VAR
	pAdress 		: PVOID;
	st_Variable		: ST_VarBuffer;
	bJson			: BOOL;
	tempString		: STRING;
	tempReal		: REAL;
	fbJson      	: FB_JsonSaxWriter;
	sJsonDocX12     : STRING(255);
	sJsonDocX11     : STRING(255);
	
	jsonKey			: STRING;
	i				: INT; // for loop index
	st_RW			: ST_RW;
END_VAR

VAR_OUTPUT
	sName			: STRING;
	eUpdate			: eUpdate;
	//bNumber		: BOOL;
	//bJson			: BOOL;
END_VAR
IF index < eDataMappingVarnames.last AND (aData[index].LogType = 0 OR aData[index].Label = '') THEN
	RETURN;
END_IF

CASE index OF 

//----(1)--- FILL STRUCTURES WITH DATA FROM PLC ------------------------------------------------------------
//----------------------------------------------------------------------------------------------------------
//--- eUpdate 0=Fast 1=Slow 2=Onchange 3=Daily--------------------------------------------------------------
//--- OnChange messages only get published when changing, at the same rate as the Fast timer----------------
//----st_Buffer contains properties of the given variable---------------------------------------------------
eDataMappingVarNames.safety_b_SafetyOK: 				st_Variable:= IotExtractType(monitor.safety.b_SafetyOK, 0, 0); 
eDataMappingVarNames.safety_b_EstopChannelAOK: 				st_Variable:= IotExtractType(monitor.safety.b_EstopChannelAOK, 0, 0); 
eDataMappingVarNames.safety_b_EstopChannelBOK: 				st_Variable:= IotExtractType(monitor.safety.b_EstopChannelBOK, 0, 0); 
eDataMappingVarNames.safety_b_InsulationMonitorOK: 				st_Variable:= IotExtractType(monitor.safety.b_InsulationMonitorOK, 0, 0); 
eDataMappingVarNames.safety_b_MRCDBOK: 				st_Variable:= IotExtractType(monitor.safety.b_MRCDBOK, 0, 0); 
// eDataMappingVarNames.safety_b_InverterDoorOK: 				st_Variable:= IotExtractType(monitor.safety.b_InverterDoorOK, 0, 0); 
// eDataMappingVarNames.safety_b_ZptOK: 				st_Variable:= IotExtractType(monitor.safety.b_ZptOK, 0, 0); 
// eDataMappingVarNames.system_b_SMSnumberConfigured: 				st_Variable:= IotExtractType(monitor.system.b_SMSnumberConfigured, 0, 0); 
// eDataMappingVarNames.system_b_CustomNameConfigured: 				st_Variable:= IotExtractType(monitor.system.b_CustomNameConfigured, 0, 0); 
// eDataMappingVarNames.system_s_SystemName: 				st_Variable:= IotExtractType(monitor.system.s_SystemName, 0, 0); 
// eDataMappingVarNames.system_b_TransportModePending: 				st_Variable:= IotExtractType(monitor.system.b_TransportModePending, 0, 0); 
// eDataMappingVarNames.system_b_DehumModePending: 				st_Variable:= IotExtractType(monitor.system.b_DehumModePending, 0, 0); 
// eDataMappingVarNames.system_e_State: 				st_Variable:= IotExtractType(monitor.system.e_State, 0, 0); 
// eDataMappingVarNames.system_e_gridmode: 				st_Variable:= IotExtractType(monitor.system.e_gridmode, 0, 0); 
// eDataMappingVarNames.system_e_UgridPowermode: 				st_Variable:= IotExtractType(monitor.system.e_UgridPowermode, 0, 0); 
// eDataMappingVarNames.system_b_StartAllowed: 				st_Variable:= IotExtractType(monitor.system.b_StartAllowed, 0, 0); 
// eDataMappingVarNames.system_r_CurrentEfficiency: 				st_Variable:= IotExtractType(monitor.system.r_CurrentEfficiency, 1, 0); 
// eDataMappingVarNames.system_r_AvgEfficiency: 				st_Variable:= IotExtractType(monitor.system.r_AvgEfficiency, 1, 0); 
// eDataMappingVarNames.system_r_RoundtripEfficiency: 				st_Variable:= IotExtractType(monitor.system.r_RoundtripEfficiency, 1, 0); 
// eDataMappingVarNames.system_DT_SystemTime: 				st_Variable:= IotExtractType(monitor.system.DT_SystemTime, 0, 0); 
// eDataMappingVarNames.system_PowerController_r_CurrentAct: 				st_Variable:= IotExtractType(monitor.system.PowerController.r_CurrentAct, 0, 1); 
// eDataMappingVarNames.system_PowerController_r_Sact: 				st_Variable:= IotExtractType(monitor.system.PowerController.r_Sact, 0, 1); 
// eDataMappingVarNames.system_PowerController_r_PAct: 				st_Variable:= IotExtractType(monitor.system.PowerController.r_PAct, 0, 1); 
// eDataMappingVarNames.system_PowerController_r_QAct: 				st_Variable:= IotExtractType(monitor.system.PowerController.r_QAct, 0, 1); 
// eDataMappingVarNames.system_PowerController_r_PhaseVoltageAct: 				st_Variable:= IotExtractType(monitor.system.PowerController.r_PhaseVoltageAct, 0, 1); 
// eDataMappingVarNames.system_PowerController_r_PFact: 				st_Variable:= IotExtractType(monitor.system.PowerController.r_PFact, 2, 0); 
// eDataMappingVarNames.system_PowerController_r_FeedInCurrentLimitActual: 				st_Variable:= IotExtractType(monitor.system.PowerController.r_FeedInCurrentLimitActual, 0, 0); 
// eDataMappingVarNames.system_PowerController_r_SupplyInCurrentLimitActual: 				st_Variable:= IotExtractType(monitor.system.PowerController.r_SupplyInCurrentLimitActual, 0, 0); 
// eDataMappingVarNames.system_PowerController_b_ThrottlingActive: 				st_Variable:= IotExtractType(monitor.system.PowerController.b_ThrottlingActive, 0, 0); 
// eDataMappingVarNames.system_PowerController_ui_ThrottlingType: 				st_Variable:= IotExtractType(monitor.system.PowerController.ui_ThrottlingType, 0, 0); 
// eDataMappingVarNames.system_PowerController_events_b_ReactivePIDError: 				st_Variable:= IotExtractType(monitor.system.PowerController.events.b_ReactivePIDError, 0, 0); 
// eDataMappingVarNames.system_PowerController_events_b_ActivePIDError: 				st_Variable:= IotExtractType(monitor.system.PowerController.events.b_ActivePIDError, 0, 0); 
// eDataMappingVarNames.system_PowerController_events_b_FreqShiftPIDError: 				st_Variable:= IotExtractType(monitor.system.PowerController.events.b_FreqShiftPIDError, 0, 0); 
// eDataMappingVarNames.system_GenGridController_b_active: 				st_Variable:= IotExtractType(monitor.system.GenGridController.b_active, 0, 0); 
// eDataMappingVarNames.system_GenGridController_b_faultActive: 				st_Variable:= IotExtractType(monitor.system.GenGridController.b_faultActive, 0, 0); 
// eDataMappingVarNames.system_GenGridController_b_gensetHot: 				st_Variable:= IotExtractType(monitor.system.GenGridController.b_gensetHot, 0, 0); 
// eDataMappingVarNames.system_GenGridController_b_gensetStarting: 				st_Variable:= IotExtractType(monitor.system.GenGridController.b_gensetStarting, 0, 0); 
// eDataMappingVarNames.system_GenGridController_b_ModeTransActive: 				st_Variable:= IotExtractType(monitor.system.GenGridController.b_ModeTransActive, 0, 0); 
// eDataMappingVarNames.system_GenGridController_b_ModeTransInhibit: 				st_Variable:= IotExtractType(monitor.system.GenGridController.b_ModeTransInhibit, 0, 0); 
// eDataMappingVarNames.system_GenGridController_b_ModeChanged: 				st_Variable:= IotExtractType(monitor.system.GenGridController.b_ModeChanged, 0, 0); 
// eDataMappingVarNames.system_GenGridController_b_ShowModeTrans: 				st_Variable:= IotExtractType(monitor.system.GenGridController.b_ShowModeTrans, 0, 0); 
// eDataMappingVarNames.system_GenGridController_b_extGensetMode: 				st_Variable:= IotExtractType(monitor.system.GenGridController.b_extGensetMode, 0, 0); 
// eDataMappingVarNames.system_GenGridController_b_gensetcontrol: 				st_Variable:= IotExtractType(monitor.system.GenGridController.b_gensetcontrol, 0, 0); 
// eDataMappingVarNames.system_GenGridController_e_BreakerMode: 				st_Variable:= IotExtractType(monitor.system.GenGridController.e_BreakerMode, 0, 0); 
// eDataMappingVarNames.system_GenGridController_e_PowerControlMode: 				st_Variable:= IotExtractType(monitor.system.GenGridController.e_PowerControlMode, 0, 0); 
// eDataMappingVarNames.system_GenGridController_e_GensetMode: 				st_Variable:= IotExtractType(monitor.system.GenGridController.e_GensetMode, 0, 0); 
// eDataMappingVarNames.system_GenGridController_e_GensetStartStop: 				st_Variable:= IotExtractType(monitor.system.GenGridController.e_GensetStartStop, 0, 0); 
// eDataMappingVarNames.system_GenGridController_e_state: 				st_Variable:= IotExtractType(monitor.system.GenGridController.e_state, 0, 0); 
// eDataMappingVarNames.system_GenGridController_e_RunCondition: 				st_Variable:= IotExtractType(monitor.system.GenGridController.e_RunCondition, 0, 0); 
// eDataMappingVarNames.system_GenGridController_events_b_InvalidGensetParameters: 				st_Variable:= IotExtractType(monitor.system.GenGridController.events.b_InvalidGensetParameters, 0, 0); 
// eDataMappingVarNames.system_GenGridController_events_b_RotationFieldFault: 				st_Variable:= IotExtractType(monitor.system.GenGridController.events.b_RotationFieldFault, 0, 0); 
// eDataMappingVarNames.system_GenGridController_events_b_CurrentLimitDisconnect: 				st_Variable:= IotExtractType(monitor.system.GenGridController.events.b_CurrentLimitDisconnect, 0, 0); 
// eDataMappingVarNames.system_GenGridController_events_b_CurrentLimitTrip: 				st_Variable:= IotExtractType(monitor.system.GenGridController.events.b_CurrentLimitTrip, 0, 0); 
// eDataMappingVarNames.system_GenGridController_events_b_EmstopDisconnect: 				st_Variable:= IotExtractType(monitor.system.GenGridController.events.b_EmstopDisconnect, 0, 0); 
// eDataMappingVarNames.system_GenGridController_events_b_ShutdownDisconnect: 				st_Variable:= IotExtractType(monitor.system.GenGridController.events.b_ShutdownDisconnect, 0, 0); 
// eDataMappingVarNames.system_GenGridController_events_b_OverloadTrip: 				st_Variable:= IotExtractType(monitor.system.GenGridController.events.b_OverloadTrip, 0, 0); 
// eDataMappingVarNames.system_GenGridController_events_b_OverFreqTrip: 				st_Variable:= IotExtractType(monitor.system.GenGridController.events.b_OverFreqTrip, 0, 0); 
// eDataMappingVarNames.system_GenGridController_events_b_UnderFreqTrip: 				st_Variable:= IotExtractType(monitor.system.GenGridController.events.b_UnderFreqTrip, 0, 0); 
// eDataMappingVarNames.system_GenGridController_events_b_OverVoltTrip: 				st_Variable:= IotExtractType(monitor.system.GenGridController.events.b_OverVoltTrip, 0, 0); 
// eDataMappingVarNames.system_GenGridController_events_b_UnderVoltTrip: 				st_Variable:= IotExtractType(monitor.system.GenGridController.events.b_UnderVoltTrip, 0, 0); 
// eDataMappingVarNames.system_GenGridController_events_b_ShutdownTimeOut: 				st_Variable:= IotExtractType(monitor.system.GenGridController.events.b_ShutdownTimeOut, 0, 0); 
// eDataMappingVarNames.system_GenGridController_events_b_SynchronisationFault: 				st_Variable:= IotExtractType(monitor.system.GenGridController.events.b_SynchronisationFault, 0, 0); 
// eDataMappingVarNames.system_GenGridController_events_b_StartupFault: 				st_Variable:= IotExtractType(monitor.system.GenGridController.events.b_StartupFault, 0, 0); 
// eDataMappingVarNames.system_GenGridController_events_b_WarmupFault: 				st_Variable:= IotExtractType(monitor.system.GenGridController.events.b_WarmupFault, 0, 0); 
// eDataMappingVarNames.system_GenGridController_events_b_GenDownTrip: 				st_Variable:= IotExtractType(monitor.system.GenGridController.events.b_GenDownTrip, 0, 0); 
// eDataMappingVarNames.system_GenGridController_events_b_GridLostTrip: 				st_Variable:= IotExtractType(monitor.system.GenGridController.events.b_GridLostTrip, 0, 0); 
// eDataMappingVarNames.system_GenGridController_events_b_TransToGenIsoInhibit: 				st_Variable:= IotExtractType(monitor.system.GenGridController.events.b_TransToGenIsoInhibit, 0, 0); 
// eDataMappingVarNames.system_GenGridController_events_b_TransToGenDroopInhibit: 				st_Variable:= IotExtractType(monitor.system.GenGridController.events.b_TransToGenDroopInhibit, 0, 0); 
// eDataMappingVarNames.system_GenGridController_events_b_TransToGenFixInhibit: 				st_Variable:= IotExtractType(monitor.system.GenGridController.events.b_TransToGenFixInhibit, 0, 0); 
// eDataMappingVarNames.system_GenGridController_events_b_TransFromInputGridAckRQ: 				st_Variable:= IotExtractType(monitor.system.GenGridController.events.b_TransFromInputGridAckRQ, 0, 0); 
// eDataMappingVarNames.system_GenGridController_events_b_TransFromInputGenAckRQ: 				st_Variable:= IotExtractType(monitor.system.GenGridController.events.b_TransFromInputGenAckRQ, 0, 0); 
// eDataMappingVarNames.system_GenGridController_events_b_StartingInhibit: 				st_Variable:= IotExtractType(monitor.system.GenGridController.events.b_StartingInhibit, 0, 0); 
// eDataMappingVarNames.system_events_b_RestartRequiredMachineName: 				st_Variable:= IotExtractType(monitor.system.events.b_RestartRequiredMachineName, 0, 0); 
// eDataMappingVarNames.system_events_b_TimeUpdateFailed: 				st_Variable:= IotExtractType(monitor.system.events.b_TimeUpdateFailed, 0, 0); 
// eDataMappingVarNames.powerstack_e_State: 				st_Variable:= IotExtractType(monitor.powerstack.e_State, 0, 0); 
// eDataMappingVarNames.powerstack_e_PowerState: 				st_Variable:= IotExtractType(monitor.powerstack.e_PowerState, 0, 0); 
// eDataMappingVarNames.powerstack_e_InverterMode: 				st_Variable:= IotExtractType(monitor.powerstack.e_InverterMode, 0, 0); 
// eDataMappingVarNames.powerstack_e_PowerMode: 				st_Variable:= IotExtractType(monitor.powerstack.e_PowerMode, 0, 0); 
// eDataMappingVarNames.powerstack_e_ThrottlingStatus: 				st_Variable:= IotExtractType(monitor.powerstack.e_ThrottlingStatus, 0, 0); 
// eDataMappingVarNames.powerstack_r_VoltageDroop: 				st_Variable:= IotExtractType(monitor.powerstack.r_VoltageDroop, 1, 0); 
// eDataMappingVarNames.powerstack_r_FrequencyDroop: 				st_Variable:= IotExtractType(monitor.powerstack.r_FrequencyDroop, 1, 0); 
// eDataMappingVarNames.powerstack_r_ACVoltageD7: 				st_Variable:= IotExtractType(monitor.powerstack.r_ACVoltageD7, 1, 1); 
// eDataMappingVarNames.powerstack_r_FrequencyD7: 				st_Variable:= IotExtractType(monitor.powerstack.r_FrequencyD7, 2, 1); 
// eDataMappingVarNames.powerstack_r_ActivePower: 				st_Variable:= IotExtractType(monitor.powerstack.r_ActivePower, 1, 1); 
// eDataMappingVarNames.powerstack_r_ReactivePower: 				st_Variable:= IotExtractType(monitor.powerstack.r_ReactivePower, 1, 1); 
// eDataMappingVarNames.powerstack_r_Pmin: 				st_Variable:= IotExtractType(monitor.powerstack.r_Pmin, 0, 0); 
// eDataMappingVarNames.powerstack_r_Pmax: 				st_Variable:= IotExtractType(monitor.powerstack.r_Pmax, 0, 0); 
// eDataMappingVarNames.powerstack_r_QMax: 				st_Variable:= IotExtractType(monitor.powerstack.r_QMax, 0, 0); 
// eDataMappingVarNames.powerstack_r_QMin: 				st_Variable:= IotExtractType(monitor.powerstack.r_QMin, 0, 0); 
// eDataMappingVarNames.powerstack_r_Smax: 				st_Variable:= IotExtractType(monitor.powerstack.r_Smax, 0, 0); 
// eDataMappingVarNames.powerstack_r_ACcurrentLimit: 				st_Variable:= IotExtractType(monitor.powerstack.r_ACcurrentLimit, 0, 0); 
// eDataMappingVarNames.powerstack_r_ACcurrentLimitMax: 				st_Variable:= IotExtractType(monitor.powerstack.r_ACcurrentLimitMax, 0, 0); 
// eDataMappingVarNames.powerstack_r_PowerChangeRate: 				st_Variable:= IotExtractType(monitor.powerstack.r_PowerChangeRate, 0, 0); 
// eDataMappingVarNames.powerstack_r_ApparentPower: 				st_Variable:= IotExtractType(monitor.powerstack.r_ApparentPower, 1, 1); 
// eDataMappingVarNames.powerstack_r_CosPhi: 				st_Variable:= IotExtractType(monitor.powerstack.r_CosPhi, 2, 0); 
// eDataMappingVarNames.powerstack_r_AcCurrent: 				st_Variable:= IotExtractType(monitor.powerstack.r_AcCurrent, 1, 0); 
// eDataMappingVarNames.powerstack_r_DCPower: 				st_Variable:= IotExtractType(monitor.powerstack.r_DCPower, 0, 1); 
// eDataMappingVarNames.powerstack_r_DCVoltage: 				st_Variable:= IotExtractType(monitor.powerstack.r_DCVoltage, 0, 1); 
// eDataMappingVarNames.powerstack_r_DCcurrent: 				st_Variable:= IotExtractType(monitor.powerstack.r_DCcurrent, 1, 1); 
// eDataMappingVarNames.powerstack_r_ACVoltageSupply: 				st_Variable:= IotExtractType(monitor.powerstack.r_ACVoltageSupply, 1, 1); 
// eDataMappingVarNames.powerstack_r_FrequencySupply: 				st_Variable:= IotExtractType(monitor.powerstack.r_FrequencySupply, 2, 1); 
// eDataMappingVarNames.powerstack_r_LoadPercent: 				st_Variable:= IotExtractType(monitor.powerstack.r_LoadPercent, 2, 0); 
// eDataMappingVarNames.powerstack_r_RatedCurrent: 				st_Variable:= IotExtractType(monitor.powerstack.r_RatedCurrent, 0, 0); 
// eDataMappingVarNames.powerstack_r_RatedPower: 				st_Variable:= IotExtractType(monitor.powerstack.r_RatedPower, 0, 0); 
// eDataMappingVarNames.powerstack_r_OvercurrentValueAct: 				st_Variable:= IotExtractType(monitor.powerstack.r_OvercurrentValueAct, 2, 0); 
// eDataMappingVarNames.powerstack_r_OvercurrentValueMax: 				st_Variable:= IotExtractType(monitor.powerstack.r_OvercurrentValueMax, 2, 0); 
// eDataMappingVarNames.powerstack_r_ThrottlingValueAct: 				st_Variable:= IotExtractType(monitor.powerstack.r_ThrottlingValueAct, 2, 0); 
// eDataMappingVarNames.powerstack_b_GridTied: 				st_Variable:= IotExtractType(monitor.powerstack.b_GridTied, 0, 0); 
// eDataMappingVarNames.powerstack_b_GridCodeCheckActive: 				st_Variable:= IotExtractType(monitor.powerstack.b_GridCodeCheckActive, 0, 0); 
// eDataMappingVarNames.powerstack_b_GridCodeOK: 				st_Variable:= IotExtractType(monitor.powerstack.b_GridCodeOK, 0, 0); 
// eDataMappingVarNames.powerstack_b_GridACdetected: 				st_Variable:= IotExtractType(monitor.powerstack.b_GridACdetected, 0, 0); 
// eDataMappingVarNames.powerstack_b_InverterGridFormingMode: 				st_Variable:= IotExtractType(monitor.powerstack.b_InverterGridFormingMode, 0, 0); 
// eDataMappingVarNames.powerstack_b_ACDetected: 				st_Variable:= IotExtractType(monitor.powerstack.b_ACDetected, 0, 0); 
// eDataMappingVarNames.powerstack_b_DCDetected: 				st_Variable:= IotExtractType(monitor.powerstack.b_DCDetected, 0, 0); 
// eDataMappingVarNames.powerstack_b_InverterRunning: 				st_Variable:= IotExtractType(monitor.powerstack.b_InverterRunning, 0, 0); 
// eDataMappingVarNames.powerstack_b_StartedState: 				st_Variable:= IotExtractType(monitor.powerstack.b_StartedState, 0, 0); 
// eDataMappingVarNames.powerstack_b_ControlEnabled: 				st_Variable:= IotExtractType(monitor.powerstack.b_ControlEnabled, 0, 0); 
// eDataMappingVarNames.powerstack_b_EcomodeAvailable: 				st_Variable:= IotExtractType(monitor.powerstack.b_EcomodeAvailable, 0, 0); 
// eDataMappingVarNames.powerstack_b_StartEnabled: 				st_Variable:= IotExtractType(monitor.powerstack.b_StartEnabled, 0, 0); 
// eDataMappingVarNames.powerstack_r_MaxTemperature: 				st_Variable:= IotExtractType(monitor.powerstack.r_MaxTemperature, 0, 0); 
// eDataMappingVarNames.powerstack_t_ShiftHoldTimeRemaining: 				st_Variable:= IotExtractType(monitor.powerstack.t_ShiftHoldTimeRemaining, 0, 0); 
// eDataMappingVarNames.powerstack_t_GridCodeReconnectTime: 				st_Variable:= IotExtractType(monitor.powerstack.t_GridCodeReconnectTime, 0, 0); 
// eDataMappingVarNames.powerstack_Events_b_CoolingDerating: 				st_Variable:= IotExtractType(monitor.powerstack.Events.b_CoolingDerating, 0, 0); 
// eDataMappingVarNames.powerstack_Events_b_PlimitShiftingActive: 				st_Variable:= IotExtractType(monitor.powerstack.Events.b_PlimitShiftingActive, 0, 0); 
// eDataMappingVarNames.powerstack_Events_b_DCdeviationHigh: 				st_Variable:= IotExtractType(monitor.powerstack.Events.b_DCdeviationHigh, 0, 0); 
// eDataMappingVarNames.powerstack_Events_b_TemperatureWarning: 				st_Variable:= IotExtractType(monitor.powerstack.Events.b_TemperatureWarning, 0, 0); 
// eDataMappingVarNames.powerstack_Events_b_OvercurrentWarning: 				st_Variable:= IotExtractType(monitor.powerstack.Events.b_OvercurrentWarning, 0, 0); 
// eDataMappingVarNames.powerstack_Events_b_UndervoltageWarning: 				st_Variable:= IotExtractType(monitor.powerstack.Events.b_UndervoltageWarning, 0, 0); 
// eDataMappingVarNames.powerstack_Events_b_OvervoltageWarning: 				st_Variable:= IotExtractType(monitor.powerstack.Events.b_OvervoltageWarning, 0, 0); 
// eDataMappingVarNames.powerstack_Events_b_TemperatureDeviationHigh: 				st_Variable:= IotExtractType(monitor.powerstack.Events.b_TemperatureDeviationHigh, 0, 0); 
// eDataMappingVarNames.powerstack_Events_b_PlimitShutdownWarning: 				st_Variable:= IotExtractType(monitor.powerstack.Events.b_PlimitShutdownWarning, 0, 0); 
// eDataMappingVarNames.powerstack_Events_b_MasterWarning: 				st_Variable:= IotExtractType(monitor.powerstack.Events.b_MasterWarning, 0, 0); 
// eDataMappingVarNames.powerstack_Events_b_SlaveWarning: 				st_Variable:= IotExtractType(monitor.powerstack.Events.b_SlaveWarning, 0, 0); 
// eDataMappingVarNames.powerstack_Events_b_GridCodeWarning: 				st_Variable:= IotExtractType(monitor.powerstack.Events.b_GridCodeWarning, 0, 0); 
// eDataMappingVarNames.powerstack_Events_b_UnderFreqFault: 				st_Variable:= IotExtractType(monitor.powerstack.Events.b_UnderFreqFault, 0, 0); 
// eDataMappingVarNames.powerstack_Events_b_OverFreqFault: 				st_Variable:= IotExtractType(monitor.powerstack.Events.b_OverFreqFault, 0, 0); 
// eDataMappingVarNames.powerstack_Events_b_UnderVoltageFault: 				st_Variable:= IotExtractType(monitor.powerstack.Events.b_UnderVoltageFault, 0, 0); 
// eDataMappingVarNames.powerstack_Events_b_OverVoltageFault: 				st_Variable:= IotExtractType(monitor.powerstack.Events.b_OverVoltageFault, 0, 0); 
// eDataMappingVarNames.powerstack_Events_b_OvercurrentFault: 				st_Variable:= IotExtractType(monitor.powerstack.Events.b_OvercurrentFault, 0, 0); 
// eDataMappingVarNames.powerstack_Events_b_PlimitShutdown: 				st_Variable:= IotExtractType(monitor.powerstack.Events.b_PlimitShutdown, 0, 0); 
// eDataMappingVarNames.powerstack_Events_b_TemperatureFault: 				st_Variable:= IotExtractType(monitor.powerstack.Events.b_TemperatureFault, 0, 0); 
// eDataMappingVarNames.powerstack_Events_b_MasterFault: 				st_Variable:= IotExtractType(monitor.powerstack.Events.b_MasterFault, 0, 0); 
// eDataMappingVarNames.powerstack_Events_b_SlaveFault: 				st_Variable:= IotExtractType(monitor.powerstack.Events.b_SlaveFault, 0, 0); 
// eDataMappingVarNames.powerstack_Events_b_NetcontactorFault: 				st_Variable:= IotExtractType(monitor.powerstack.Events.b_NetcontactorFault, 0, 0); 
// eDataMappingVarNames.powerstack_Events_b_startupTimeOut: 				st_Variable:= IotExtractType(monitor.powerstack.Events.b_startupTimeOut, 0, 0); 
// eDataMappingVarNames.powerstack_Events_b_ShutdownTimeOut: 				st_Variable:= IotExtractType(monitor.powerstack.Events.b_ShutdownTimeOut, 0, 0); 
// eDataMappingVarNames.powerstack_Events_ui_shutdownRemainingTime: 				st_Variable:= IotExtractType(monitor.powerstack.Events.ui_shutdownRemainingTime, 0, 0); 
// eDataMappingVarNames.powerstack_PowermoduleMaster_b_online: 				st_Variable:= IotExtractType(monitor.powerstack.PowermoduleMaster.b_online, 0, 0); 
// eDataMappingVarNames.powerstack_PowermoduleMaster_r_ApparentPower: 				st_Variable:= IotExtractType(monitor.powerstack.PowermoduleMaster.r_ApparentPower, 0, 1); 
// eDataMappingVarNames.powerstack_PowermoduleMaster_r_ActivePower: 				st_Variable:= IotExtractType(monitor.powerstack.PowermoduleMaster.r_ActivePower, 1, 1); 
// eDataMappingVarNames.powerstack_PowermoduleMaster_r_ReactivePower: 				st_Variable:= IotExtractType(monitor.powerstack.PowermoduleMaster.r_ReactivePower, 1, 1); 
// eDataMappingVarNames.powerstack_PowermoduleMaster_r_ACVoltageD7: 				st_Variable:= IotExtractType(monitor.powerstack.PowermoduleMaster.r_ACVoltageD7, 1, 1); 
// eDataMappingVarNames.powerstack_PowermoduleMaster_r_VoltageDroop: 				st_Variable:= IotExtractType(monitor.powerstack.PowermoduleMaster.r_VoltageDroop, 1, 0); 
// eDataMappingVarNames.powerstack_PowermoduleMaster_r_ACVoltageSupply: 				st_Variable:= IotExtractType(monitor.powerstack.PowermoduleMaster.r_ACVoltageSupply, 1, 1); 
// eDataMappingVarNames.powerstack_PowermoduleMaster_r_FrequencyD7: 				st_Variable:= IotExtractType(monitor.powerstack.PowermoduleMaster.r_FrequencyD7, 1, 1); 
// eDataMappingVarNames.powerstack_PowermoduleMaster_r_FrequencyDroop: 				st_Variable:= IotExtractType(monitor.powerstack.PowermoduleMaster.r_FrequencyDroop, 1, 0); 
// eDataMappingVarNames.powerstack_PowermoduleMaster_r_FrequencySupply: 				st_Variable:= IotExtractType(monitor.powerstack.PowermoduleMaster.r_FrequencySupply, 2, 1); 
// eDataMappingVarNames.powerstack_PowermoduleMaster_r_CurrentUnbalance: 				st_Variable:= IotExtractType(monitor.powerstack.PowermoduleMaster.r_CurrentUnbalance, 1, 1); 
// eDataMappingVarNames.powerstack_PowermoduleMaster_r_DCPower: 				st_Variable:= IotExtractType(monitor.powerstack.PowermoduleMaster.r_DCPower, 0, 1); 
// eDataMappingVarNames.powerstack_PowermoduleMaster_r_DCVoltage: 				st_Variable:= IotExtractType(monitor.powerstack.PowermoduleMaster.r_DCVoltage, 0, 1); 
// eDataMappingVarNames.powerstack_PowermoduleMaster_r_DCCurrent: 				st_Variable:= IotExtractType(monitor.powerstack.PowermoduleMaster.r_DCCurrent, 1, 0); 
// eDataMappingVarNames.powerstack_PowermoduleMaster_r_ACCurrent: 				st_Variable:= IotExtractType(monitor.powerstack.PowermoduleMaster.r_ACCurrent, 1, 1); 
// eDataMappingVarNames.powerstack_PowermoduleMaster_r_ActiveCurrent: 				st_Variable:= IotExtractType(monitor.powerstack.PowermoduleMaster.r_ActiveCurrent, 1, 1); 
// eDataMappingVarNames.powerstack_PowermoduleMaster_r_ReactiveCurrent: 				st_Variable:= IotExtractType(monitor.powerstack.PowermoduleMaster.r_ReactiveCurrent, 1, 1); 
// eDataMappingVarNames.powerstack_PowermoduleMaster_r_LoadPercent: 				st_Variable:= IotExtractType(monitor.powerstack.PowermoduleMaster.r_LoadPercent, 1, 0); 
// eDataMappingVarNames.powerstack_PowermoduleMaster_r_D7SyncError: 				st_Variable:= IotExtractType(monitor.powerstack.PowermoduleMaster.r_D7SyncError, 1, 0); 
// eDataMappingVarNames.powerstack_PowermoduleMaster_r_Pmin: 				st_Variable:= IotExtractType(monitor.powerstack.PowermoduleMaster.r_Pmin, 0, 0); 
// eDataMappingVarNames.powerstack_PowermoduleMaster_r_Pmax: 				st_Variable:= IotExtractType(monitor.powerstack.PowermoduleMaster.r_Pmax, 0, 0); 
// eDataMappingVarNames.powerstack_PowermoduleMaster_r_QMax: 				st_Variable:= IotExtractType(monitor.powerstack.PowermoduleMaster.r_QMax, 0, 0); 
// eDataMappingVarNames.powerstack_PowermoduleMaster_r_Qmin: 				st_Variable:= IotExtractType(monitor.powerstack.PowermoduleMaster.r_Qmin, 0, 0); 
// eDataMappingVarNames.powerstack_PowermoduleMaster_r_Pset: 				st_Variable:= IotExtractType(monitor.powerstack.PowermoduleMaster.r_Pset, 0, 0); 
// eDataMappingVarNames.powerstack_PowermoduleMaster_r_Qset: 				st_Variable:= IotExtractType(monitor.powerstack.PowermoduleMaster.r_Qset, 0, 0); 
// eDataMappingVarNames.powerstack_PowermoduleMaster_r_ACcurrentLimit: 				st_Variable:= IotExtractType(monitor.powerstack.PowermoduleMaster.r_ACcurrentLimit, 0, 0); 
// eDataMappingVarNames.powerstack_PowermoduleMaster_r_OverCurrentValue: 				st_Variable:= IotExtractType(monitor.powerstack.PowermoduleMaster.r_OverCurrentValue, 2, 0); 
// eDataMappingVarNames.powerstack_PowermoduleMaster_r_ModulationIndex: 				st_Variable:= IotExtractType(monitor.powerstack.PowermoduleMaster.r_ModulationIndex, 2, 0); 
// eDataMappingVarNames.powerstack_PowermoduleMaster_r_TemperatureInverter: 				st_Variable:= IotExtractType(monitor.powerstack.PowermoduleMaster.r_TemperatureInverter, 1, 0); 
// eDataMappingVarNames.powerstack_PowermoduleMaster_r_TemperatureGridChoke_1: 				st_Variable:= IotExtractType(monitor.powerstack.PowermoduleMaster.r_TemperatureGridChoke[1], 1, 0); 
// eDataMappingVarNames.powerstack_PowermoduleMaster_r_TemperatureGridChoke_2: 				st_Variable:= IotExtractType(monitor.powerstack.PowermoduleMaster.r_TemperatureGridChoke[2], 1, 0); 
// eDataMappingVarNames.powerstack_PowermoduleMaster_r_TemperatureGridChoke_3: 				st_Variable:= IotExtractType(monitor.powerstack.PowermoduleMaster.r_TemperatureGridChoke[3], 1, 0); 
// eDataMappingVarNames.powerstack_PowermoduleMaster_r_TemperatureCMChoke_1: 				st_Variable:= IotExtractType(monitor.powerstack.PowermoduleMaster.r_TemperatureCMChoke[1], 1, 0); 
// eDataMappingVarNames.powerstack_PowermoduleMaster_r_TemperatureCMChoke_2: 				st_Variable:= IotExtractType(monitor.powerstack.PowermoduleMaster.r_TemperatureCMChoke[2], 1, 0); 
// eDataMappingVarNames.powerstack_PowermoduleMaster_r_TemperatureCMChoke_3: 				st_Variable:= IotExtractType(monitor.powerstack.PowermoduleMaster.r_TemperatureCMChoke[3], 1, 0); 
// eDataMappingVarNames.powerstack_PowermoduleMaster_r_TemperatureCMChoke_4: 				st_Variable:= IotExtractType(monitor.powerstack.PowermoduleMaster.r_TemperatureCMChoke[4], 1, 0); 
// eDataMappingVarNames.powerstack_PowermoduleMaster_r_TemperatureMax: 				st_Variable:= IotExtractType(monitor.powerstack.PowermoduleMaster.r_TemperatureMax, 1, 0); 
// eDataMappingVarNames.powerstack_PowermoduleSlave_w_TemperatureFaultWord: 				st_Variable:= IotExtractType(monitor.powerstack.PowermoduleSlave.w_TemperatureFaultWord, 0, 0); 
// eDataMappingVarNames.powerstack_PowermoduleSlave_w_OperationHours: 				st_Variable:= IotExtractType(monitor.powerstack.PowermoduleSlave.w_OperationHours, 0, 0); 
// eDataMappingVarNames.powerstack_PowermoduleSlave_e_PowerMode: 				st_Variable:= IotExtractType(monitor.powerstack.PowermoduleSlave.e_PowerMode, 0, 0); 
// eDataMappingVarNames.powerstack_PowermoduleSlave_e_InverterMode: 				st_Variable:= IotExtractType(monitor.powerstack.PowermoduleSlave.e_InverterMode, 0, 0); 
// eDataMappingVarNames.powerstack_PowermoduleSlave_e_Status: 				st_Variable:= IotExtractType(monitor.powerstack.PowermoduleSlave.e_Status, 0, 0); 
// eDataMappingVarNames.powerstack_PowermoduleSlave_e_ThrottlingStatus: 				st_Variable:= IotExtractType(monitor.powerstack.PowermoduleSlave.e_ThrottlingStatus, 0, 0); 
// eDataMappingVarNames.powerstack_PowermoduleSlave_ui_InverterCommStatus: 				st_Variable:= IotExtractType(monitor.powerstack.PowermoduleSlave.ui_InverterCommStatus, 0, 0); 
// eDataMappingVarNames.powerstack_PowermoduleSlave_ui_BuscouplerCommStatus: 				st_Variable:= IotExtractType(monitor.powerstack.PowermoduleSlave.ui_BuscouplerCommStatus, 0, 0); 
// eDataMappingVarNames.powerstack_PowermoduleSlave_b_MccbTripOK: 				st_Variable:= IotExtractType(monitor.powerstack.PowermoduleSlave.b_MccbTripOK, 0, 0); 
// eDataMappingVarNames.powerstack_PowermoduleSlave_b_MccbUvr24VdcOK: 				st_Variable:= IotExtractType(monitor.powerstack.PowermoduleSlave.b_MccbUvr24VdcOK, 0, 0); 
// eDataMappingVarNames.powerstack_PowermoduleSlave_b_MccbFb: 				st_Variable:= IotExtractType(monitor.powerstack.PowermoduleSlave.b_MccbFb, 0, 0); 
// eDataMappingVarNames.powerstack_PowermoduleSlave_b_FanFb: 				st_Variable:= IotExtractType(monitor.powerstack.PowermoduleSlave.b_FanFb, 0, 0); 
// eDataMappingVarNames.powerstack_PowermoduleSlave_b_DCcontactorFb: 				st_Variable:= IotExtractType(monitor.powerstack.PowermoduleSlave.b_DCcontactorFb, 0, 0); 
// eDataMappingVarNames.powerstack_PowermoduleSlave_b_PrechargeContactor: 				st_Variable:= IotExtractType(monitor.powerstack.PowermoduleSlave.b_PrechargeContactor, 0, 0); 
// eDataMappingVarNames.powerstack_PowermoduleSlave_b_LimiterActive: 				st_Variable:= IotExtractType(monitor.powerstack.PowermoduleSlave.b_LimiterActive, 0, 0); 
// eDataMappingVarNames.powerstack_PowermoduleSlave_StatusWord_b_ReadyToDCCharge: 				st_Variable:= IotExtractType(monitor.powerstack.PowermoduleSlave.StatusWord.b_ReadyToDCCharge, 0, 0); 
// eDataMappingVarNames.powerstack_PowermoduleSlave_StatusWord_b_ReadyToOperate: 				st_Variable:= IotExtractType(monitor.powerstack.PowermoduleSlave.StatusWord.b_ReadyToOperate, 0, 0); 
// eDataMappingVarNames.powerstack_PowermoduleSlave_StatusWord_b_Running: 				st_Variable:= IotExtractType(monitor.powerstack.PowermoduleSlave.StatusWord.b_Running, 0, 0); 
// eDataMappingVarNames.powerstack_PowermoduleSlave_StatusWord_b_Fault: 				st_Variable:= IotExtractType(monitor.powerstack.PowermoduleSlave.StatusWord.b_Fault, 0, 0); 
// eDataMappingVarNames.powerstack_PowermoduleSlave_StatusWord_b_RunEnabled: 				st_Variable:= IotExtractType(monitor.powerstack.PowermoduleSlave.StatusWord.b_RunEnabled, 0, 0); 
// eDataMappingVarNames.powerstack_PowermoduleSlave_StatusWord_b_QuickstopNotActive: 				st_Variable:= IotExtractType(monitor.powerstack.PowermoduleSlave.StatusWord.b_QuickstopNotActive, 0, 0); 
// eDataMappingVarNames.powerstack_PowermoduleSlave_StatusWord_b_MCCBControlNotOK: 				st_Variable:= IotExtractType(monitor.powerstack.PowermoduleSlave.StatusWord.b_MCCBControlNotOK, 0, 0); 
// eDataMappingVarNames.powerstack_PowermoduleSlave_StatusWord_b_Warning: 				st_Variable:= IotExtractType(monitor.powerstack.PowermoduleSlave.StatusWord.b_Warning, 0, 0); 
// eDataMappingVarNames.powerstack_PowermoduleSlave_StatusWord_b_DCAtReference: 				st_Variable:= IotExtractType(monitor.powerstack.PowermoduleSlave.StatusWord.b_DCAtReference, 0, 0); 
// eDataMappingVarNames.powerstack_PowermoduleSlave_StatusWord_b_DCAboveLimit: 				st_Variable:= IotExtractType(monitor.powerstack.PowermoduleSlave.StatusWord.b_DCAboveLimit, 0, 0); 
// eDataMappingVarNames.powerstack_PowermoduleSlave_StatusWord_b_WatchdogFeedback: 				st_Variable:= IotExtractType(monitor.powerstack.PowermoduleSlave.StatusWord.b_WatchdogFeedback, 0, 0); 
// eDataMappingVarNames.powerstack_PowermoduleSlave_UgridStatusWord_b_ChargeControlActive: 				st_Variable:= IotExtractType(monitor.powerstack.PowermoduleSlave.UgridStatusWord.b_ChargeControlActive, 0, 0); 
// eDataMappingVarNames.powerstack_PowermoduleSlave_UgridStatusWord_b_InternalChargingSwitchStatus: 				st_Variable:= IotExtractType(monitor.powerstack.PowermoduleSlave.UgridStatusWord.b_InternalChargingSwitchStatus, 0, 0); 
// eDataMappingVarNames.powerstack_PowermoduleSlave_UgridStatusWord_b_MCBcontrol: 				st_Variable:= IotExtractType(monitor.powerstack.PowermoduleSlave.UgridStatusWord.b_MCBcontrol, 0, 0); 
// eDataMappingVarNames.powerstack_PowermoduleSlave_UgridStatusWord_b_MCBStatus: 				st_Variable:= IotExtractType(monitor.powerstack.PowermoduleSlave.UgridStatusWord.b_MCBStatus, 0, 0); 
// eDataMappingVarNames.powerstack_PowermoduleSlave_UgridStatusWord_b_RunEnabled: 				st_Variable:= IotExtractType(monitor.powerstack.PowermoduleSlave.UgridStatusWord.b_RunEnabled, 0, 0); 
// eDataMappingVarNames.powerstack_PowermoduleSlave_UgridStatusWord_b_DriveReady: 				st_Variable:= IotExtractType(monitor.powerstack.PowermoduleSlave.UgridStatusWord.b_DriveReady, 0, 0); 
// eDataMappingVarNames.powerstack_PowermoduleSlave_UgridStatusWord_b_AFEmodeActive: 				st_Variable:= IotExtractType(monitor.powerstack.PowermoduleSlave.UgridStatusWord.b_AFEmodeActive, 0, 0); 
// eDataMappingVarNames.powerstack_PowermoduleSlave_UgridStatusWord_b_IslandModeActive: 				st_Variable:= IotExtractType(monitor.powerstack.PowermoduleSlave.UgridStatusWord.b_IslandModeActive, 0, 0); 
// eDataMappingVarNames.powerstack_PowermoduleSlave_UgridStatusWord_b_MicrogridModeActive: 				st_Variable:= IotExtractType(monitor.powerstack.PowermoduleSlave.UgridStatusWord.b_MicrogridModeActive, 0, 0); 
// eDataMappingVarNames.powerstack_PowermoduleSlave_UgridStatusWord_b_RunRequestActive: 				st_Variable:= IotExtractType(monitor.powerstack.PowermoduleSlave.UgridStatusWord.b_RunRequestActive, 0, 0); 
// eDataMappingVarNames.powerstack_PowermoduleSlave_UgridStatusWord_b_DriveInRunState: 				st_Variable:= IotExtractType(monitor.powerstack.PowermoduleSlave.UgridStatusWord.b_DriveInRunState, 0, 0); 
// eDataMappingVarNames.powerstack_PowermoduleSlave_UgridStatusWord_b_FaultActive: 				st_Variable:= IotExtractType(monitor.powerstack.PowermoduleSlave.UgridStatusWord.b_FaultActive, 0, 0); 
// eDataMappingVarNames.powerstack_PowermoduleSlave_UgridStatusWord_b_SynchronizedToD7: 				st_Variable:= IotExtractType(monitor.powerstack.PowermoduleSlave.UgridStatusWord.b_SynchronizedToD7, 0, 0); 
// eDataMappingVarNames.powerstack_PowermoduleSlave_UgridStatusWord_b_D7MeasurementsOK: 				st_Variable:= IotExtractType(monitor.powerstack.PowermoduleSlave.UgridStatusWord.b_D7MeasurementsOK, 0, 0); 
// eDataMappingVarNames.powerstack_PowermoduleSlave_GridcodeStatusWord_b_LineVoltTripLimHigh: 				st_Variable:= IotExtractType(monitor.powerstack.PowermoduleSlave.GridcodeStatusWord.b_LineVoltTripLimHigh, 0, 0); 
// eDataMappingVarNames.powerstack_PowermoduleSlave_GridcodeStatusWord_b_LineVoltTripLimlow: 				st_Variable:= IotExtractType(monitor.powerstack.PowermoduleSlave.GridcodeStatusWord.b_LineVoltTripLimlow, 0, 0); 
// eDataMappingVarNames.powerstack_PowermoduleSlave_GridcodeStatusWord_b_LineFreqTripLimHigh: 				st_Variable:= IotExtractType(monitor.powerstack.PowermoduleSlave.GridcodeStatusWord.b_LineFreqTripLimHigh, 0, 0); 
// eDataMappingVarNames.powerstack_PowermoduleSlave_GridcodeStatusWord_b_LineFreqTripLimLow: 				st_Variable:= IotExtractType(monitor.powerstack.PowermoduleSlave.GridcodeStatusWord.b_LineFreqTripLimLow, 0, 0); 
// eDataMappingVarNames.powerstack_PowermoduleSlave_GridcodeStatusWord_b_LineFreqOK: 				st_Variable:= IotExtractType(monitor.powerstack.PowermoduleSlave.GridcodeStatusWord.b_LineFreqOK, 0, 0); 
// eDataMappingVarNames.powerstack_PowermoduleSlave_GridcodeStatusWord_b_LineVoltOK: 				st_Variable:= IotExtractType(monitor.powerstack.PowermoduleSlave.GridcodeStatusWord.b_LineVoltOK, 0, 0); 
// eDataMappingVarNames.powerstack_PowermoduleSlave_GridcodeStatusWord_b_FRTActive: 				st_Variable:= IotExtractType(monitor.powerstack.PowermoduleSlave.GridcodeStatusWord.b_FRTActive, 0, 0); 
// eDataMappingVarNames.powerstack_PowermoduleSlave_GridcodeStatusWord_b_GridCodeTripActive: 				st_Variable:= IotExtractType(monitor.powerstack.PowermoduleSlave.GridcodeStatusWord.b_GridCodeTripActive, 0, 0); 
// eDataMappingVarNames.powerstack_PowermoduleSlave_Events_b_GeneralFaultFlag: 				st_Variable:= IotExtractType(monitor.powerstack.PowermoduleSlave.Events.b_GeneralFaultFlag, 0, 0); 
// eDataMappingVarNames.powerstack_PowermoduleSlave_Events_b_GeneralWarningFlag: 				st_Variable:= IotExtractType(monitor.powerstack.PowermoduleSlave.Events.b_GeneralWarningFlag, 0, 0); 
// eDataMappingVarNames.powerstack_PowermoduleSlave_Events_b_CMSTemperatureRangeWarning: 				st_Variable:= IotExtractType(monitor.powerstack.PowermoduleSlave.Events.b_CMSTemperatureRangeWarning, 0, 0); 
// eDataMappingVarNames.powerstack_PowermoduleSlave_Events_b_FanStateUnknownWarning: 				st_Variable:= IotExtractType(monitor.powerstack.PowermoduleSlave.Events.b_FanStateUnknownWarning, 0, 0); 
// eDataMappingVarNames.powerstack_PowermoduleSlave_Events_b_TempThrottlingActive: 				st_Variable:= IotExtractType(monitor.powerstack.PowermoduleSlave.Events.b_TempThrottlingActive, 0, 0); 
// eDataMappingVarNames.powerstack_PowermoduleSlave_Events_b_CurrThrottlingActive: 				st_Variable:= IotExtractType(monitor.powerstack.PowermoduleSlave.Events.b_CurrThrottlingActive, 0, 0); 
// eDataMappingVarNames.powerstack_PowermoduleSlave_Events_b_F1OverCurrent: 				st_Variable:= IotExtractType(monitor.powerstack.PowermoduleSlave.Events.b_F1OverCurrent, 0, 0); 
// eDataMappingVarNames.powerstack_PowermoduleSlave_Events_b_F2OverVoltage: 				st_Variable:= IotExtractType(monitor.powerstack.PowermoduleSlave.Events.b_F2OverVoltage, 0, 0); 
// eDataMappingVarNames.powerstack_PowermoduleSlave_Events_b_F9UnderVoltage: 				st_Variable:= IotExtractType(monitor.powerstack.PowermoduleSlave.Events.b_F9UnderVoltage, 0, 0); 
// eDataMappingVarNames.powerstack_PowermoduleSlave_Events_b_F91ShortCircuit: 				st_Variable:= IotExtractType(monitor.powerstack.PowermoduleSlave.Events.b_F91ShortCircuit, 0, 0); 
// eDataMappingVarNames.powerstack_PowermoduleSlave_Events_b_F3EarthFault: 				st_Variable:= IotExtractType(monitor.powerstack.PowermoduleSlave.Events.b_F3EarthFault, 0, 0); 
// eDataMappingVarNames.powerstack_PowermoduleSlave_Events_b_Spare: 				st_Variable:= IotExtractType(monitor.powerstack.PowermoduleSlave.Events.b_Spare, 0, 0); 
// eDataMappingVarNames.powerstack_PowermoduleSlave_Events_b_F14UnitOverTemperature: 				st_Variable:= IotExtractType(monitor.powerstack.PowermoduleSlave.Events.b_F14UnitOverTemperature, 0, 0); 
// eDataMappingVarNames.powerstack_PowermoduleSlave_Events_b_F56TemperatureFault: 				st_Variable:= IotExtractType(monitor.powerstack.PowermoduleSlave.Events.b_F56TemperatureFault, 0, 0); 
// eDataMappingVarNames.powerstack_PowermoduleSlave_Events_b_F10LineSynchFault: 				st_Variable:= IotExtractType(monitor.powerstack.PowermoduleSlave.Events.b_F10LineSynchFault, 0, 0); 
// eDataMappingVarNames.powerstack_PowermoduleSlave_Events_b_F52KeypadOCCommFault: 				st_Variable:= IotExtractType(monitor.powerstack.PowermoduleSlave.Events.b_F52KeypadOCCommFault, 0, 0); 
// eDataMappingVarNames.powerstack_PowermoduleSlave_Events_b_F53FieldbusFault: 				st_Variable:= IotExtractType(monitor.powerstack.PowermoduleSlave.Events.b_F53FieldbusFault, 0, 0); 
// eDataMappingVarNames.powerstack_PowermoduleSlave_Events_b_F59SystembusFault: 				st_Variable:= IotExtractType(monitor.powerstack.PowermoduleSlave.Events.b_F59SystembusFault, 0, 0); 
// eDataMappingVarNames.powerstack_PowermoduleSlave_Events_b_F54SlotCommunicationFault: 				st_Variable:= IotExtractType(monitor.powerstack.PowermoduleSlave.Events.b_F54SlotCommunicationFault, 0, 0); 
// eDataMappingVarNames.powerstack_PowermoduleSlave_Events_b_F50Meas4mAFault: 				st_Variable:= IotExtractType(monitor.powerstack.PowermoduleSlave.Events.b_F50Meas4mAFault, 0, 0); 
// eDataMappingVarNames.powerstack_PowermoduleSlave_Events_b_F11OutputPhaseFault: 				st_Variable:= IotExtractType(monitor.powerstack.PowermoduleSlave.Events.b_F11OutputPhaseFault, 0, 0); 
// eDataMappingVarNames.powerstack_PowermoduleSlave_Events_b_F80ChargeFault: 				st_Variable:= IotExtractType(monitor.powerstack.PowermoduleSlave.Events.b_F80ChargeFault, 0, 0); 
// eDataMappingVarNames.powerstack_PowermoduleSlave_Events_b_F51ExternalFault: 				st_Variable:= IotExtractType(monitor.powerstack.PowermoduleSlave.Events.b_F51ExternalFault, 0, 0); 
// eDataMappingVarNames.powerstack_PowermoduleSlave_Events_b_F31IGBTFault: 				st_Variable:= IotExtractType(monitor.powerstack.PowermoduleSlave.Events.b_F31IGBTFault, 0, 0); 
// eDataMappingVarNames.powerstack_PowermoduleSlave_Events_b_F64MCBstateFault: 				st_Variable:= IotExtractType(monitor.powerstack.PowermoduleSlave.Events.b_F64MCBstateFault, 0, 0); 
// eDataMappingVarNames.powerstack_PowermoduleSlave_Events_b_WatchdogError: 				st_Variable:= IotExtractType(monitor.powerstack.PowermoduleSlave.Events.b_WatchdogError, 0, 0); 
// eDataMappingVarNames.powerstack_PowermoduleSlave_Events_b_24VdcUVRFault: 				st_Variable:= IotExtractType(monitor.powerstack.PowermoduleSlave.Events.b_24VdcUVRFault, 0, 0); 
// eDataMappingVarNames.powerstack_PowermoduleSlave_Events_b_MCCBtrip: 				st_Variable:= IotExtractType(monitor.powerstack.PowermoduleSlave.Events.b_MCCBtrip, 0, 0); 
// eDataMappingVarNames.powerstack_PowermoduleSlave_Events_b_ShutdownTimeOut: 				st_Variable:= IotExtractType(monitor.powerstack.PowermoduleSlave.Events.b_ShutdownTimeOut, 0, 0); 
// eDataMappingVarNames.powerstack_PowermoduleSlave_Events_b_StartUpTimeOut: 				st_Variable:= IotExtractType(monitor.powerstack.PowermoduleSlave.Events.b_StartUpTimeOut, 0, 0); 
// eDataMappingVarNames.powerstack_PowermoduleSlave_Events_b_CMChokeTemperatureHigh_1: 				st_Variable:= IotExtractType(monitor.powerstack.PowermoduleSlave.Events.b_CMChokeTemperatureHigh[1], 0, 0); 
// eDataMappingVarNames.powerstack_PowermoduleSlave_Events_b_CMChokeTemperatureHigh_2: 				st_Variable:= IotExtractType(monitor.powerstack.PowermoduleSlave.Events.b_CMChokeTemperatureHigh[2], 0, 0); 
// eDataMappingVarNames.powerstack_PowermoduleSlave_Events_b_CMChokeTemperatureHigh_3: 				st_Variable:= IotExtractType(monitor.powerstack.PowermoduleSlave.Events.b_CMChokeTemperatureHigh[3], 0, 0); 
// eDataMappingVarNames.powerstack_PowermoduleSlave_Events_b_CMChokeTemperatureHigh_4: 				st_Variable:= IotExtractType(monitor.powerstack.PowermoduleSlave.Events.b_CMChokeTemperatureHigh[4], 0, 0); 
// eDataMappingVarNames.powerstack_PowermoduleSlave_Events_b_CMChokeTemperatureTooHigh_1: 				st_Variable:= IotExtractType(monitor.powerstack.PowermoduleSlave.Events.b_CMChokeTemperatureTooHigh[1], 0, 0); 
// eDataMappingVarNames.powerstack_PowermoduleSlave_Events_b_CMChokeTemperatureTooHigh_2: 				st_Variable:= IotExtractType(monitor.powerstack.PowermoduleSlave.Events.b_CMChokeTemperatureTooHigh[2], 0, 0); 
// eDataMappingVarNames.powerstack_PowermoduleSlave_Events_b_CMChokeTemperatureTooHigh_3: 				st_Variable:= IotExtractType(monitor.powerstack.PowermoduleSlave.Events.b_CMChokeTemperatureTooHigh[3], 0, 0); 
// eDataMappingVarNames.powerstack_PowermoduleSlave_Events_b_CMChokeTemperatureTooHigh_4: 				st_Variable:= IotExtractType(monitor.powerstack.PowermoduleSlave.Events.b_CMChokeTemperatureTooHigh[4], 0, 0); 
// eDataMappingVarNames.powerstack_PowermoduleSlave_Events_b_GridChokeTemperatureHigh_1: 				st_Variable:= IotExtractType(monitor.powerstack.PowermoduleSlave.Events.b_GridChokeTemperatureHigh[1], 0, 0); 
// eDataMappingVarNames.powerstack_PowermoduleSlave_Events_b_GridChokeTemperatureHigh_2: 				st_Variable:= IotExtractType(monitor.powerstack.PowermoduleSlave.Events.b_GridChokeTemperatureHigh[2], 0, 0); 
// eDataMappingVarNames.powerstack_PowermoduleSlave_Events_b_GridChokeTemperatureHigh_3: 				st_Variable:= IotExtractType(monitor.powerstack.PowermoduleSlave.Events.b_GridChokeTemperatureHigh[3], 0, 0); 
// eDataMappingVarNames.powerstack_PowermoduleSlave_Events_b_GridChokeTemperatureTooHigh_1: 				st_Variable:= IotExtractType(monitor.powerstack.PowermoduleSlave.Events.b_GridChokeTemperatureTooHigh[1], 0, 0); 
// eDataMappingVarNames.powerstack_PowermoduleSlave_Events_b_GridChokeTemperatureTooHigh_2: 				st_Variable:= IotExtractType(monitor.powerstack.PowermoduleSlave.Events.b_GridChokeTemperatureTooHigh[2], 0, 0); 
// eDataMappingVarNames.powerstack_PowermoduleSlave_Events_b_GridChokeTemperatureTooHigh_3: 				st_Variable:= IotExtractType(monitor.powerstack.PowermoduleSlave.Events.b_GridChokeTemperatureTooHigh[3], 0, 0); 
// eDataMappingVarNames.powerstack_PowermoduleSlave_Events_b_inverterTemperatureHigh: 				st_Variable:= IotExtractType(monitor.powerstack.PowermoduleSlave.Events.b_inverterTemperatureHigh, 0, 0); 
// eDataMappingVarNames.powerstack_PowermoduleSlave_Events_b_PT100Overrange: 				st_Variable:= IotExtractType(monitor.powerstack.PowermoduleSlave.Events.b_PT100Overrange, 0, 0); 
// eDataMappingVarNames.powerstack_PowermoduleSlave_Events_b_PT100Underrange: 				st_Variable:= IotExtractType(monitor.powerstack.PowermoduleSlave.Events.b_PT100Underrange, 0, 0); 
// eDataMappingVarNames.powerstack_PowermoduleSlave_Events_by_PT100ErrorCount: 				st_Variable:= IotExtractType(monitor.powerstack.PowermoduleSlave.Events.by_PT100ErrorCount, 0, 0); 
// eDataMappingVarNames.powerstack_PowermoduleSlave_controldata_Controlword_b_ChargeDC: 				st_Variable:= IotExtractType(monitor.powerstack.PowermoduleSlave.controldata.Controlword.b_ChargeDC, 0, 0); 
// eDataMappingVarNames.powerstack_PowermoduleSlave_controldata_Controlword_b_run: 				st_Variable:= IotExtractType(monitor.powerstack.PowermoduleSlave.controldata.Controlword.b_run, 0, 0); 
// eDataMappingVarNames.powerstack_PowermoduleSlave_controldata_Controlword_b_Reset: 				st_Variable:= IotExtractType(monitor.powerstack.PowermoduleSlave.controldata.Controlword.b_Reset, 0, 0); 
// eDataMappingVarNames.powerstack_PowermoduleSlave_controldata_Controlword_b_FieldbusControlEnable: 				st_Variable:= IotExtractType(monitor.powerstack.PowermoduleSlave.controldata.Controlword.b_FieldbusControlEnable, 0, 0); 
// eDataMappingVarNames.powerstack_PowermoduleSlave_controldata_Controlword_b_WatchdogPulse: 				st_Variable:= IotExtractType(monitor.powerstack.PowermoduleSlave.controldata.Controlword.b_WatchdogPulse, 0, 0); 
// eDataMappingVarNames.powerstack_PowermoduleSlave_controldata_Controlword_b_ParallelAFE: 				st_Variable:= IotExtractType(monitor.powerstack.PowermoduleSlave.controldata.Controlword.b_ParallelAFE, 0, 0); 
// eDataMappingVarNames.powerstack_PowermoduleSlave_controldata_Controlword_b_PIDenable: 				st_Variable:= IotExtractType(monitor.powerstack.PowermoduleSlave.controldata.Controlword.b_PIDenable, 0, 0); 
// eDataMappingVarNames.powerstack_PowermoduleSlave_controldata_Controlword_b_GridCodeEnable: 				st_Variable:= IotExtractType(monitor.powerstack.PowermoduleSlave.controldata.Controlword.b_GridCodeEnable, 0, 0); 
// eDataMappingVarNames.powerstack_PowermoduleSlave_controldata_Controlword_b_ExtGridcodeTrip: 				st_Variable:= IotExtractType(monitor.powerstack.PowermoduleSlave.controldata.Controlword.b_ExtGridcodeTrip, 0, 0); 
// eDataMappingVarNames.powerstack_PowermoduleSlave_controldata_ui_ControlwordValue: 				st_Variable:= IotExtractType(monitor.powerstack.PowermoduleSlave.controldata.ui_ControlwordValue, 0, 0); 
// eDataMappingVarNames.powerstack_PowermoduleSlave_controldata_i_invertermode: 				st_Variable:= IotExtractType(monitor.powerstack.PowermoduleSlave.controldata.i_invertermode, 0, 0); 
// eDataMappingVarNames.powerstack_PowermoduleSlave_controldata_i_BaseCurrentRef: 				st_Variable:= IotExtractType(monitor.powerstack.PowermoduleSlave.controldata.i_BaseCurrentRef, 0, 0); 
// eDataMappingVarNames.powerstack_PowermoduleSlave_controldata_i_ReactiveCurrentRef: 				st_Variable:= IotExtractType(monitor.powerstack.PowermoduleSlave.controldata.i_ReactiveCurrentRef, 0, 0); 
// eDataMappingVarNames.powerstack_PowermoduleSlave_controldata_i_FrequencyDroop: 				st_Variable:= IotExtractType(monitor.powerstack.PowermoduleSlave.controldata.i_FrequencyDroop, 0, 0); 
// eDataMappingVarNames.powerstack_PowermoduleSlave_controldata_i_VoltageDroop: 				st_Variable:= IotExtractType(monitor.powerstack.PowermoduleSlave.controldata.i_VoltageDroop, 0, 0); 
// eDataMappingVarNames.powerstack_PowermoduleSlave_controldata_i_FrequencyDroopOffset: 				st_Variable:= IotExtractType(monitor.powerstack.PowermoduleSlave.controldata.i_FrequencyDroopOffset, 0, 0); 
// eDataMappingVarNames.powerstack_PowermoduleSlave_controldata_i_VoltageCorrection: 				st_Variable:= IotExtractType(monitor.powerstack.PowermoduleSlave.controldata.i_VoltageCorrection, 0, 0); 
// eDataMappingVarNames.powerstack_PowermoduleSlave_controldata_i_BaseRefRampRate: 				st_Variable:= IotExtractType(monitor.powerstack.PowermoduleSlave.controldata.i_BaseRefRampRate, 0, 0); 
// eDataMappingVarNames.powerstack_PowermoduleSlave_controldata_i_StartPowerMode: 				st_Variable:= IotExtractType(monitor.powerstack.PowermoduleSlave.controldata.i_StartPowerMode, 0, 0); 
// eDataMappingVarNames.powerstack_PowermoduleSlave_controldata_i_StartVoltageMode: 				st_Variable:= IotExtractType(monitor.powerstack.PowermoduleSlave.controldata.i_StartVoltageMode, 0, 0); 
// eDataMappingVarNames.powerstack_PowermoduleSlave_controldata_i_OutActCurrentLimit: 				st_Variable:= IotExtractType(monitor.powerstack.PowermoduleSlave.controldata.i_OutActCurrentLimit, 0, 0); 
// eDataMappingVarNames.powerstack_PowermoduleSlave_controldata_i_InActCurrentLimit: 				st_Variable:= IotExtractType(monitor.powerstack.PowermoduleSlave.controldata.i_InActCurrentLimit, 0, 0); 
// eDataMappingVarNames.powerstack_PowermoduleSlave_controldata_i_DCVramprate: 				st_Variable:= IotExtractType(monitor.powerstack.PowermoduleSlave.controldata.i_DCVramprate, 0, 0); 
// eDataMappingVarNames.powerstack_Netcontactor_e_NetConState: 				st_Variable:= IotExtractType(monitor.powerstack.Netcontactor.e_NetConState, 0, 0); 
// eDataMappingVarNames.powerstack_Netcontactor_b_SyncCloseCommand: 				st_Variable:= IotExtractType(monitor.powerstack.Netcontactor.b_SyncCloseCommand, 0, 0); 
// eDataMappingVarNames.powerstack_Netcontactor_b_NetConFb: 				st_Variable:= IotExtractType(monitor.powerstack.Netcontactor.b_NetConFb, 0, 0); 
// eDataMappingVarNames.powerstack_Netcontactor_b_NetcontRightFb: 				st_Variable:= IotExtractType(monitor.powerstack.Netcontactor.b_NetcontRightFb, 0, 0); 
// eDataMappingVarNames.powerstack_Netcontactor_b_NetcontLeftFb: 				st_Variable:= IotExtractType(monitor.powerstack.Netcontactor.b_NetcontLeftFb, 0, 0); 
// eDataMappingVarNames.powerstack_Netcontactor_events_b_AMFEnabled: 				st_Variable:= IotExtractType(monitor.powerstack.Netcontactor.events.b_AMFEnabled, 0, 0); 
// eDataMappingVarNames.powerstack_Netcontactor_events_b_ContactorRightFbFault: 				st_Variable:= IotExtractType(monitor.powerstack.Netcontactor.events.b_ContactorRightFbFault, 0, 0); 
// eDataMappingVarNames.powerstack_Netcontactor_events_b_ContactorLeftFbFault: 				st_Variable:= IotExtractType(monitor.powerstack.Netcontactor.events.b_ContactorLeftFbFault, 0, 0); 
// eDataMappingVarNames.powerstack_Netcontactor_events_b_ContactorFbTimeout: 				st_Variable:= IotExtractType(monitor.powerstack.Netcontactor.events.b_ContactorFbTimeout, 0, 0); 
// eDataMappingVarNames.powerstack_Netcontactor_events_b_PhaseRotationFault: 				st_Variable:= IotExtractType(monitor.powerstack.Netcontactor.events.b_PhaseRotationFault, 0, 0); 
// eDataMappingVarNames.powerstack_Netcontactor_events_b_IllegalLeftFieldSelected: 				st_Variable:= IotExtractType(monitor.powerstack.Netcontactor.events.b_IllegalLeftFieldSelected, 0, 0); 
// eDataMappingVarNames.powermonitor_PQMeterReady: 								st_Variable:= IotExtractType(monitor.powermonitor.PQMeterReady, 0, 0); 
// eDataMappingVarNames.powermonitor_InputField_ar_ApparentPower_AVG: 				st_Variable:= IotExtractType(monitor.powermonitor.InputField.ar_ApparentPower[0], 1, 1); 
// eDataMappingVarNames.powermonitor_InputField_ar_ApparentPower_L1: 				st_Variable:= IotExtractType(monitor.powermonitor.InputField.ar_ApparentPower[1], 1, 1); 
// eDataMappingVarNames.powermonitor_InputField_ar_ApparentPower_L2: 				st_Variable:= IotExtractType(monitor.powermonitor.InputField.ar_ApparentPower[2], 1, 1); 
// eDataMappingVarNames.powermonitor_InputField_ar_ApparentPower_L3: 				st_Variable:= IotExtractType(monitor.powermonitor.InputField.ar_ApparentPower[3], 1, 1); 
// eDataMappingVarNames.powermonitor_InputField_ar_ReactivePower_AVG: 				st_Variable:= IotExtractType(monitor.powermonitor.InputField.ar_ReactivePower[0], 1, 1); 
// eDataMappingVarNames.powermonitor_InputField_ar_ReactivePower_L1: 				st_Variable:= IotExtractType(monitor.powermonitor.InputField.ar_ReactivePower[1], 1, 1); 
// eDataMappingVarNames.powermonitor_InputField_ar_ReactivePower_L2: 				st_Variable:= IotExtractType(monitor.powermonitor.InputField.ar_ReactivePower[2], 1, 1); 
// eDataMappingVarNames.powermonitor_InputField_ar_ReactivePower_L3: 				st_Variable:= IotExtractType(monitor.powermonitor.InputField.ar_ReactivePower[3], 1, 1); 
// eDataMappingVarNames.powermonitor_InputField_ar_ActivePower_AVG: 				st_Variable:= IotExtractType(monitor.powermonitor.InputField.ar_ActivePower[0], 1, 1); 
// eDataMappingVarNames.powermonitor_InputField_ar_ActivePower_L1: 				st_Variable:= IotExtractType(monitor.powermonitor.InputField.ar_ActivePower[1], 1, 1); 
// eDataMappingVarNames.powermonitor_InputField_ar_ActivePower_L2: 				st_Variable:= IotExtractType(monitor.powermonitor.InputField.ar_ActivePower[2], 1, 1); 
// eDataMappingVarNames.powermonitor_InputField_ar_ActivePower_L3: 				st_Variable:= IotExtractType(monitor.powermonitor.InputField.ar_ActivePower[3], 1, 1); 
// eDataMappingVarNames.powermonitor_InputField_r_EnergyConsumed: 				st_Variable:= IotExtractType(monitor.powermonitor.InputField.r_EnergyConsumed, 0, 0); 
// eDataMappingVarNames.powermonitor_InputField_r_EnergySupplied: 				st_Variable:= IotExtractType(monitor.powermonitor.InputField.r_EnergySupplied, 0, 0); 
// eDataMappingVarNames.powermonitor_InputField_ar_THD_AVG: 				st_Variable:= IotExtractType(monitor.powermonitor.InputField.ar_THD[0], 1, 0); 
// eDataMappingVarNames.powermonitor_InputField_ar_THD_L1: 				st_Variable:= IotExtractType(monitor.powermonitor.InputField.ar_THD[1], 1, 0); 
// eDataMappingVarNames.powermonitor_InputField_ar_THD_L2: 				st_Variable:= IotExtractType(monitor.powermonitor.InputField.ar_THD[2], 1, 0); 
// eDataMappingVarNames.powermonitor_InputField_ar_THD_L3: 				st_Variable:= IotExtractType(monitor.powermonitor.InputField.ar_THD[3], 1, 0); 
// eDataMappingVarNames.powermonitor_InputField_ar_PowerFactor_AVG: 				st_Variable:= IotExtractType(monitor.powermonitor.InputField.ar_PowerFactor[0], 2, 0); 
// eDataMappingVarNames.powermonitor_InputField_ar_PowerFactor_L1: 				st_Variable:= IotExtractType(monitor.powermonitor.InputField.ar_PowerFactor[1], 2, 0); 
// eDataMappingVarNames.powermonitor_InputField_ar_PowerFactor_L2: 				st_Variable:= IotExtractType(monitor.powermonitor.InputField.ar_PowerFactor[2], 2, 0); 
// eDataMappingVarNames.powermonitor_InputField_ar_PowerFactor_L3: 				st_Variable:= IotExtractType(monitor.powermonitor.InputField.ar_PowerFactor[3], 2, 0); 
// eDataMappingVarNames.powermonitor_InputField_ar_Current_AVG: 				st_Variable:= IotExtractType(monitor.powermonitor.InputField.ar_Current[0], 0, 1); 
// eDataMappingVarNames.powermonitor_InputField_ar_Current_L1: 				st_Variable:= IotExtractType(monitor.powermonitor.InputField.ar_Current[1], 0, 1); 
// eDataMappingVarNames.powermonitor_InputField_ar_Current_L2: 				st_Variable:= IotExtractType(monitor.powermonitor.InputField.ar_Current[2], 0, 1); 
// eDataMappingVarNames.powermonitor_InputField_ar_Current_L3: 				st_Variable:= IotExtractType(monitor.powermonitor.InputField.ar_Current[3], 0, 1); 
// eDataMappingVarNames.powermonitor_InputField_ar_Current_N: 					st_Variable:= IotExtractType(monitor.powermonitor.InputField.ar_Current[4], 0, 1); 
// eDataMappingVarNames.powermonitor_InputField_r_CurrentUnbalance: 				st_Variable:= IotExtractType(monitor.powermonitor.InputField.r_CurrentUnbalance, 1, 0); 
// eDataMappingVarNames.powermonitor_InputField_e_ACrotationStatus: 				st_Variable:= IotExtractType(monitor.powermonitor.InputField.e_ACrotationStatus, 0, 0); 
// eDataMappingVarNames.powermonitor_InputField_ar_PhaseVoltage_AVG: 				st_Variable:= IotExtractType(monitor.powermonitor.InputField.ar_PhaseVoltage[0], 1, 1); 
// eDataMappingVarNames.powermonitor_InputField_ar_PhaseVoltage_L1: 				st_Variable:= IotExtractType(monitor.powermonitor.InputField.ar_PhaseVoltage[1], 1, 1); 
// eDataMappingVarNames.powermonitor_InputField_ar_PhaseVoltage_L2: 				st_Variable:= IotExtractType(monitor.powermonitor.InputField.ar_PhaseVoltage[2], 1, 1); 
// eDataMappingVarNames.powermonitor_InputField_ar_PhaseVoltage_L3: 				st_Variable:= IotExtractType(monitor.powermonitor.InputField.ar_PhaseVoltage[3], 1, 1); 
// eDataMappingVarNames.powermonitor_InputField_ar_LineVoltage_AVG: 				st_Variable:= IotExtractType(monitor.powermonitor.InputField.ar_LineVoltage[0], 1, 1); 
// eDataMappingVarNames.powermonitor_InputField_ar_LineVoltage_L1: 				st_Variable:= IotExtractType(monitor.powermonitor.InputField.ar_LineVoltage[1], 1, 1); 
// eDataMappingVarNames.powermonitor_InputField_ar_LineVoltage_L2: 				st_Variable:= IotExtractType(monitor.powermonitor.InputField.ar_LineVoltage[2], 1, 1); 
// eDataMappingVarNames.powermonitor_InputField_ar_LineVoltage_L3: 				st_Variable:= IotExtractType(monitor.powermonitor.InputField.ar_LineVoltage[3], 1, 1); 
// eDataMappingVarNames.powermonitor_InputField_li_TimeVoltZeroCrossup: 				st_Variable:= IotExtractType(monitor.powermonitor.InputField.li_TimeVoltZeroCrossup, 0, 0); 
// eDataMappingVarNames.powermonitor_InputField_ar_Frequency_AVG: 				st_Variable:= IotExtractType(monitor.powermonitor.InputField.ar_Frequency[0], 2, 1); 
// eDataMappingVarNames.powermonitor_InputField_ar_Frequency_L1: 				st_Variable:= IotExtractType(monitor.powermonitor.InputField.ar_Frequency[1], 2, 1); 
// eDataMappingVarNames.powermonitor_InputField_ar_Frequency_L2: 				st_Variable:= IotExtractType(monitor.powermonitor.InputField.ar_Frequency[2], 2, 1); 
// eDataMappingVarNames.powermonitor_InputField_ar_Frequency_L3: 				st_Variable:= IotExtractType(monitor.powermonitor.InputField.ar_Frequency[3], 2, 1); 
// eDataMappingVarNames.powermonitor_InputField_r_VoltageUnbalance: 				st_Variable:= IotExtractType(monitor.powermonitor.InputField.r_VoltageUnbalance, 1, 0); 
// eDataMappingVarNames.powermonitor_InputField_r_loadshare: 				st_Variable:= IotExtractType(monitor.powermonitor.InputField.r_loadshare, 1, 0); 
// eDataMappingVarNames.powermonitor_InputField_Powerlock_1_ar_ApparentPower_AVG: 				st_Variable:= IotExtractType(monitor.powermonitor.InputField.Powerlock[1].ar_ApparentPower[0], 0, 0); 
// eDataMappingVarNames.powermonitor_InputField_Powerlock_2_ar_ApparentPower_AVG: 				st_Variable:= IotExtractType(monitor.powermonitor.InputField.Powerlock[2].ar_ApparentPower[0], 0, 0); 
// eDataMappingVarNames.powermonitor_InputField_Powerlock_1_ar_ApparentPower_L1: 				st_Variable:= IotExtractType(monitor.powermonitor.InputField.Powerlock[1].ar_ApparentPower[1], 0, 0); 
// eDataMappingVarNames.powermonitor_InputField_Powerlock_2_ar_ApparentPower_L1: 				st_Variable:= IotExtractType(monitor.powermonitor.InputField.Powerlock[2].ar_ApparentPower[1], 0, 0); 
// eDataMappingVarNames.powermonitor_InputField_Powerlock_1_ar_ApparentPower_L2: 				st_Variable:= IotExtractType(monitor.powermonitor.InputField.Powerlock[1].ar_ApparentPower[2], 0, 0); 
// eDataMappingVarNames.powermonitor_InputField_Powerlock_2_ar_ApparentPower_L2: 				st_Variable:= IotExtractType(monitor.powermonitor.InputField.Powerlock[2].ar_ApparentPower[2], 0, 0); 
// eDataMappingVarNames.powermonitor_InputField_Powerlock_1_ar_ApparentPower_L3: 				st_Variable:= IotExtractType(monitor.powermonitor.InputField.Powerlock[1].ar_ApparentPower[3], 0, 0); 
// eDataMappingVarNames.powermonitor_InputField_Powerlock_2_ar_ApparentPower_L3: 				st_Variable:= IotExtractType(monitor.powermonitor.InputField.Powerlock[2].ar_ApparentPower[3], 0, 0); 
// eDataMappingVarNames.powermonitor_InputField_Powerlock_1_ar_ReactivePower_AVG: 				st_Variable:= IotExtractType(monitor.powermonitor.InputField.Powerlock[1].ar_ReactivePower[0], 0, 0); 
// eDataMappingVarNames.powermonitor_InputField_Powerlock_2_ar_ReactivePower_AVG: 				st_Variable:= IotExtractType(monitor.powermonitor.InputField.Powerlock[2].ar_ReactivePower[0], 0, 0); 
// eDataMappingVarNames.powermonitor_InputField_Powerlock_1_ar_ReactivePower_L1: 				st_Variable:= IotExtractType(monitor.powermonitor.InputField.Powerlock[1].ar_ReactivePower[1], 0, 0); 
// eDataMappingVarNames.powermonitor_InputField_Powerlock_2_ar_ReactivePower_L1: 				st_Variable:= IotExtractType(monitor.powermonitor.InputField.Powerlock[2].ar_ReactivePower[1], 0, 0); 
// eDataMappingVarNames.powermonitor_InputField_Powerlock_1_ar_ReactivePower_L2: 				st_Variable:= IotExtractType(monitor.powermonitor.InputField.Powerlock[1].ar_ReactivePower[2], 0, 0); 
// eDataMappingVarNames.powermonitor_InputField_Powerlock_2_ar_ReactivePower_L2: 				st_Variable:= IotExtractType(monitor.powermonitor.InputField.Powerlock[2].ar_ReactivePower[2], 0, 0); 
// eDataMappingVarNames.powermonitor_InputField_Powerlock_1_ar_ReactivePower_L3: 				st_Variable:= IotExtractType(monitor.powermonitor.InputField.Powerlock[1].ar_ReactivePower[3], 0, 0); 
// eDataMappingVarNames.powermonitor_InputField_Powerlock_2_ar_ReactivePower_L3: 				st_Variable:= IotExtractType(monitor.powermonitor.InputField.Powerlock[2].ar_ReactivePower[3], 0, 0); 
// eDataMappingVarNames.powermonitor_InputField_Powerlock_1_ar_ActivePower_AVG: 				st_Variable:= IotExtractType(monitor.powermonitor.InputField.Powerlock[1].ar_ActivePower[0]	, 0, 0); 
// eDataMappingVarNames.powermonitor_InputField_Powerlock_2_ar_ActivePower_AVG: 				st_Variable:= IotExtractType(monitor.powermonitor.InputField.Powerlock[2].ar_ActivePower[0]	, 0, 0); 
// eDataMappingVarNames.powermonitor_InputField_Powerlock_1_ar_ActivePower_L1: 				st_Variable:= IotExtractType(monitor.powermonitor.InputField.Powerlock[1].ar_ActivePower[1]	, 0, 0); 
// eDataMappingVarNames.powermonitor_InputField_Powerlock_2_ar_ActivePower_L1: 				st_Variable:= IotExtractType(monitor.powermonitor.InputField.Powerlock[2].ar_ActivePower[1]	, 0, 0); 
// eDataMappingVarNames.powermonitor_InputField_Powerlock_1_ar_ActivePower_L2: 				st_Variable:= IotExtractType(monitor.powermonitor.InputField.Powerlock[1].ar_ActivePower[2]	, 0, 0); 
// eDataMappingVarNames.powermonitor_InputField_Powerlock_2_ar_ActivePower_L2: 				st_Variable:= IotExtractType(monitor.powermonitor.InputField.Powerlock[2].ar_ActivePower[2]	, 0, 0); 
// eDataMappingVarNames.powermonitor_InputField_Powerlock_1_ar_ActivePower_L3: 				st_Variable:= IotExtractType(monitor.powermonitor.InputField.Powerlock[1].ar_ActivePower[3]	, 0, 0); 
// eDataMappingVarNames.powermonitor_InputField_Powerlock_2_ar_ActivePower_L3: 				st_Variable:= IotExtractType(monitor.powermonitor.InputField.Powerlock[2].ar_ActivePower[3]	, 0, 0); 
// eDataMappingVarNames.powermonitor_InputField_Powerlock_1_r_EnergyConsumed: 				st_Variable:= IotExtractType(monitor.powermonitor.InputField.Powerlock[1].r_EnergyConsumed, 0, 	0); 
// eDataMappingVarNames.powermonitor_InputField_Powerlock_2_r_EnergyConsumed: 				st_Variable:= IotExtractType(monitor.powermonitor.InputField.Powerlock[2].r_EnergyConsumed, 0, 	0); 
// eDataMappingVarNames.powermonitor_InputField_Powerlock_1_r_EnergySupplied: 				st_Variable:= IotExtractType(monitor.powermonitor.InputField.Powerlock[1].r_EnergySupplied, 0, 	0); 
// eDataMappingVarNames.powermonitor_InputField_Powerlock_2_r_EnergySupplied: 				st_Variable:= IotExtractType(monitor.powermonitor.InputField.Powerlock[2].r_EnergySupplied, 0, 	0); 
// eDataMappingVarNames.powermonitor_InputField_Powerlock_1_ar_THD_AVG: 				st_Variable:= IotExtractType(monitor.powermonitor.InputField.Powerlock[1].ar_THD[0], 0, 0);        	
// eDataMappingVarNames.powermonitor_InputField_Powerlock_2_ar_THD_AVG: 				st_Variable:= IotExtractType(monitor.powermonitor.InputField.Powerlock[2].ar_THD[0], 0, 0);        	
// eDataMappingVarNames.powermonitor_InputField_Powerlock_1_ar_THD_L1: 				st_Variable:= IotExtractType(monitor.powermonitor.InputField.Powerlock[1].ar_THD[1], 0, 0);        	
// eDataMappingVarNames.powermonitor_InputField_Powerlock_2_ar_THD_L1: 				st_Variable:= IotExtractType(monitor.powermonitor.InputField.Powerlock[2].ar_THD[1], 0, 0);        	
// eDataMappingVarNames.powermonitor_InputField_Powerlock_1_ar_THD_L2: 				st_Variable:= IotExtractType(monitor.powermonitor.InputField.Powerlock[1].ar_THD[2], 0, 0);        	
// eDataMappingVarNames.powermonitor_InputField_Powerlock_2_ar_THD_L2: 				st_Variable:= IotExtractType(monitor.powermonitor.InputField.Powerlock[2].ar_THD[2], 0, 0);        	
// eDataMappingVarNames.powermonitor_InputField_Powerlock_1_ar_THD_L3: 				st_Variable:= IotExtractType(monitor.powermonitor.InputField.Powerlock[1].ar_THD[3], 0, 0);        	
// eDataMappingVarNames.powermonitor_InputField_Powerlock_2_ar_THD_L3: 				st_Variable:= IotExtractType(monitor.powermonitor.InputField.Powerlock[2].ar_THD[3], 0, 0);        	
// eDataMappingVarNames.powermonitor_InputField_Powerlock_1_ar_PowerFactor_AVG: 				st_Variable:= IotExtractType(monitor.powermonitor.InputField.Powerlock[1].ar_PowerFactor[0]	, 2, 0); 
// eDataMappingVarNames.powermonitor_InputField_Powerlock_2_ar_PowerFactor_AVG: 				st_Variable:= IotExtractType(monitor.powermonitor.InputField.Powerlock[2].ar_PowerFactor[0]	, 2, 0); 
// eDataMappingVarNames.powermonitor_InputField_Powerlock_1_ar_PowerFactor_L1: 				st_Variable:= IotExtractType(monitor.powermonitor.InputField.Powerlock[1].ar_PowerFactor[1]	, 2, 0); 
// eDataMappingVarNames.powermonitor_InputField_Powerlock_2_ar_PowerFactor_L1: 				st_Variable:= IotExtractType(monitor.powermonitor.InputField.Powerlock[2].ar_PowerFactor[1]	, 2, 0); 
// eDataMappingVarNames.powermonitor_InputField_Powerlock_1_ar_PowerFactor_L2: 				st_Variable:= IotExtractType(monitor.powermonitor.InputField.Powerlock[1].ar_PowerFactor[2]	, 2, 0); 
// eDataMappingVarNames.powermonitor_InputField_Powerlock_2_ar_PowerFactor_L2: 				st_Variable:= IotExtractType(monitor.powermonitor.InputField.Powerlock[2].ar_PowerFactor[2]	, 2, 0); 
// eDataMappingVarNames.powermonitor_InputField_Powerlock_1_ar_PowerFactor_L3: 				st_Variable:= IotExtractType(monitor.powermonitor.InputField.Powerlock[1].ar_PowerFactor[3]	, 2, 0); 
// eDataMappingVarNames.powermonitor_InputField_Powerlock_2_ar_PowerFactor_L3: 				st_Variable:= IotExtractType(monitor.powermonitor.InputField.Powerlock[2].ar_PowerFactor[3]	, 2, 0); 
// eDataMappingVarNames.powermonitor_InputField_Powerlock_1_ar_Current_AVG: 				st_Variable:= IotExtractType(monitor.powermonitor.InputField.Powerlock[1].ar_Current[0]			, 1, 1); 
// eDataMappingVarNames.powermonitor_InputField_Powerlock_2_ar_Current_AVG: 				st_Variable:= IotExtractType(monitor.powermonitor.InputField.Powerlock[2].ar_Current[0]			, 1, 1); 
// eDataMappingVarNames.powermonitor_InputField_Powerlock_1_ar_Current_L1: 				st_Variable:= IotExtractType(monitor.powermonitor.InputField.Powerlock[1].ar_Current[1]			, 1, 1); 
// eDataMappingVarNames.powermonitor_InputField_Powerlock_2_ar_Current_L1: 				st_Variable:= IotExtractType(monitor.powermonitor.InputField.Powerlock[2].ar_Current[1]			, 1, 1); 
// eDataMappingVarNames.powermonitor_InputField_Powerlock_1_ar_Current_L2: 				st_Variable:= IotExtractType(monitor.powermonitor.InputField.Powerlock[1].ar_Current[2]			, 1, 1); 
// eDataMappingVarNames.powermonitor_InputField_Powerlock_2_ar_Current_L2: 				st_Variable:= IotExtractType(monitor.powermonitor.InputField.Powerlock[2].ar_Current[2]			, 1, 1); 
// eDataMappingVarNames.powermonitor_InputField_Powerlock_1_ar_Current_L3: 				st_Variable:= IotExtractType(monitor.powermonitor.InputField.Powerlock[1].ar_Current[3]			, 1, 1); 
// eDataMappingVarNames.powermonitor_InputField_Powerlock_2_ar_Current_L3: 				st_Variable:= IotExtractType(monitor.powermonitor.InputField.Powerlock[2].ar_Current[3]			, 1, 1); 
// eDataMappingVarNames.powermonitor_InputField_Powerlock_1_ar_Current_N: 				st_Variable:= IotExtractType(monitor.powermonitor.InputField.Powerlock[1].ar_Current[4], 1, 1); 
// eDataMappingVarNames.powermonitor_InputField_Powerlock_2_ar_Current_N: 				st_Variable:= IotExtractType(monitor.powermonitor.InputField.Powerlock[2].ar_Current[4], 1, 1); 
// eDataMappingVarNames.powermonitor_InputField_Powerlock_1_r_CurrentUnbalance: 				st_Variable:= IotExtractType(monitor.powermonitor.InputField.Powerlock[1].r_CurrentUnbalance, 0, 0); 
// eDataMappingVarNames.powermonitor_InputField_Powerlock_2_r_CurrentUnbalance: 				st_Variable:= IotExtractType(monitor.powermonitor.InputField.Powerlock[2].r_CurrentUnbalance, 0, 0); 
// eDataMappingVarNames.powermonitor_OutputField_ar_ApparentPower_AVG: 				st_Variable:= IotExtractType(monitor.powermonitor.OutputField.ar_ApparentPower[0]	, 1, 1); 
// eDataMappingVarNames.powermonitor_OutputField_ar_ApparentPower_L1: 				st_Variable:= IotExtractType(monitor.powermonitor.OutputField.ar_ApparentPower[1]		, 1, 1); 
// eDataMappingVarNames.powermonitor_OutputField_ar_ApparentPower_L2: 				st_Variable:= IotExtractType(monitor.powermonitor.OutputField.ar_ApparentPower[2]		, 1, 1); 
// eDataMappingVarNames.powermonitor_OutputField_ar_ApparentPower_L3: 				st_Variable:= IotExtractType(monitor.powermonitor.OutputField.ar_ApparentPower[3]		, 1, 1); 
// eDataMappingVarNames.powermonitor_OutputField_ar_ReactivePower_AVG: 				st_Variable:= IotExtractType(monitor.powermonitor.OutputField.ar_ReactivePower[0]	, 1, 1); 
// eDataMappingVarNames.powermonitor_OutputField_ar_ReactivePower_L1: 				st_Variable:= IotExtractType(monitor.powermonitor.OutputField.ar_ReactivePower[1]		, 1, 1); 
// eDataMappingVarNames.powermonitor_OutputField_ar_ReactivePower_L2: 				st_Variable:= IotExtractType(monitor.powermonitor.OutputField.ar_ReactivePower[2]		, 1, 1); 
// eDataMappingVarNames.powermonitor_OutputField_ar_ReactivePower_L3: 				st_Variable:= IotExtractType(monitor.powermonitor.OutputField.ar_ReactivePower[3]		, 1, 1); 
// eDataMappingVarNames.powermonitor_OutputField_ar_ActivePower_AVG: 				st_Variable:= IotExtractType(monitor.powermonitor.OutputField.ar_ActivePower[0]			, 1, 1); 
// eDataMappingVarNames.powermonitor_OutputField_ar_ActivePower_L1: 				st_Variable:= IotExtractType(monitor.powermonitor.OutputField.ar_ActivePower[1]			, 1, 1); 
// eDataMappingVarNames.powermonitor_OutputField_ar_ActivePower_L2: 				st_Variable:= IotExtractType(monitor.powermonitor.OutputField.ar_ActivePower[2]			, 1, 1); 
// eDataMappingVarNames.powermonitor_OutputField_ar_ActivePower_L3: 				st_Variable:= IotExtractType(monitor.powermonitor.OutputField.ar_ActivePower[3]			, 1, 1); 
// eDataMappingVarNames.powermonitor_OutputField_r_EnergyConsumed: 				st_Variable:= IotExtractType(monitor.powermonitor.OutputField.r_EnergyConsumed, 0, 0); 
// eDataMappingVarNames.powermonitor_OutputField_r_EnergySupplied: 				st_Variable:= IotExtractType(monitor.powermonitor.OutputField.r_EnergySupplied, 0, 0); 
// eDataMappingVarNames.powermonitor_OutputField_ar_THD_AVG: 				st_Variable:= IotExtractType(monitor.powermonitor.OutputField.ar_THD[0], 1, 0); 
// eDataMappingVarNames.powermonitor_OutputField_ar_THD_L1: 				st_Variable:= IotExtractType(monitor.powermonitor.OutputField.ar_THD[1], 1, 0); 
// eDataMappingVarNames.powermonitor_OutputField_ar_THD_L2: 				st_Variable:= IotExtractType(monitor.powermonitor.OutputField.ar_THD[2], 1, 0); 
// eDataMappingVarNames.powermonitor_OutputField_ar_THD_L3: 				st_Variable:= IotExtractType(monitor.powermonitor.OutputField.ar_THD[3], 1, 0); 
// eDataMappingVarNames.powermonitor_OutputField_ar_PowerFactor_AVG: 				st_Variable:= IotExtractType(monitor.powermonitor.OutputField.ar_PowerFactor[0], 2, 0); 
// eDataMappingVarNames.powermonitor_OutputField_ar_PowerFactor_L1: 				st_Variable:= IotExtractType(monitor.powermonitor.OutputField.ar_PowerFactor[1], 2, 0); 
// eDataMappingVarNames.powermonitor_OutputField_ar_PowerFactor_L2: 				st_Variable:= IotExtractType(monitor.powermonitor.OutputField.ar_PowerFactor[2], 2, 0); 
// eDataMappingVarNames.powermonitor_OutputField_ar_PowerFactor_L3: 				st_Variable:= IotExtractType(monitor.powermonitor.OutputField.ar_PowerFactor[3], 2, 0); 
// eDataMappingVarNames.powermonitor_OutputField_ar_Current_AVG: 				st_Variable:= IotExtractType(monitor.powermonitor.OutputField.ar_Current[0], 1, 1); 
// eDataMappingVarNames.powermonitor_OutputField_ar_Current_L1: 				st_Variable:= IotExtractType(monitor.powermonitor.OutputField.ar_Current[1], 1, 1); 
// eDataMappingVarNames.powermonitor_OutputField_ar_Current_L2: 				st_Variable:= IotExtractType(monitor.powermonitor.OutputField.ar_Current[2], 1, 1); 
// eDataMappingVarNames.powermonitor_OutputField_ar_Current_L3: 				st_Variable:= IotExtractType(monitor.powermonitor.OutputField.ar_Current[3], 1, 1); 
// eDataMappingVarNames.powermonitor_OutputField_ar_Current_N: 				st_Variable:= IotExtractType(monitor.powermonitor.OutputField.ar_Current[4], 1, 1); 
// eDataMappingVarNames.powermonitor_OutputField_r_CurrentUnbalance: 				st_Variable:= IotExtractType(monitor.powermonitor.OutputField.r_CurrentUnbalance, 1, 0); 
// eDataMappingVarNames.powermonitor_OutputField_e_ACrotationStatus: 				st_Variable:= IotExtractType(monitor.powermonitor.OutputField.e_ACrotationStatus, 0, 0); 
// eDataMappingVarNames.powermonitor_OutputField_ar_PhaseVoltage_AVG: 				st_Variable:= IotExtractType(monitor.powermonitor.OutputField.ar_PhaseVoltage[0], 1, 1); 
// eDataMappingVarNames.powermonitor_OutputField_ar_PhaseVoltage_L1: 				st_Variable:= IotExtractType(monitor.powermonitor.OutputField.ar_PhaseVoltage[1], 1, 1); 
// eDataMappingVarNames.powermonitor_OutputField_ar_PhaseVoltage_L2: 				st_Variable:= IotExtractType(monitor.powermonitor.OutputField.ar_PhaseVoltage[2], 1, 1); 
// eDataMappingVarNames.powermonitor_OutputField_ar_PhaseVoltage_L3: 				st_Variable:= IotExtractType(monitor.powermonitor.OutputField.ar_PhaseVoltage[3], 1, 1); 
// eDataMappingVarNames.powermonitor_OutputField_ar_LineVoltage_AVG: 				st_Variable:= IotExtractType(monitor.powermonitor.OutputField.ar_LineVoltage[0]	, 1, 1); 
// eDataMappingVarNames.powermonitor_OutputField_ar_LineVoltage_L1: 				st_Variable:= IotExtractType(monitor.powermonitor.OutputField.ar_LineVoltage[1]	, 1, 1); 
// eDataMappingVarNames.powermonitor_OutputField_ar_LineVoltage_L2: 				st_Variable:= IotExtractType(monitor.powermonitor.OutputField.ar_LineVoltage[2]	, 1, 1); 
// eDataMappingVarNames.powermonitor_OutputField_ar_LineVoltage_L3: 				st_Variable:= IotExtractType(monitor.powermonitor.OutputField.ar_LineVoltage[3]	, 1, 1); 
// eDataMappingVarNames.powermonitor_OutputField_li_TimeVoltZeroCrossup: 				st_Variable:= IotExtractType(monitor.powermonitor.OutputField.li_TimeVoltZeroCrossup, 0, 0); 
// eDataMappingVarNames.powermonitor_OutputField_ar_Frequency_AVG: 				st_Variable:= IotExtractType(monitor.powermonitor.OutputField.ar_Frequency[0], 2, 1); 
// eDataMappingVarNames.powermonitor_OutputField_ar_Frequency_L1: 				st_Variable:= IotExtractType(monitor.powermonitor.OutputField.ar_Frequency[1], 2, 1); 
// eDataMappingVarNames.powermonitor_OutputField_ar_Frequency_L2: 				st_Variable:= IotExtractType(monitor.powermonitor.OutputField.ar_Frequency[2], 2, 1); 
// eDataMappingVarNames.powermonitor_OutputField_ar_Frequency_L3: 				st_Variable:= IotExtractType(monitor.powermonitor.OutputField.ar_Frequency[3], 2, 1); 
// eDataMappingVarNames.powermonitor_OutputField_r_VoltageUnbalance: 				st_Variable:= IotExtractType(monitor.powermonitor.OutputField.r_VoltageUnbalance, 1, 0); 
// eDataMappingVarNames.powermonitor_OutputField_r_loadshare: 				st_Variable:= IotExtractType(monitor.powermonitor.OutputField.r_loadshare, 1, 0); 
// eDataMappingVarNames.powermonitor_OutputField_Powerlock_1_ar_ApparentPower_AVG: 				st_Variable:= IotExtractType(monitor.powermonitor.OutputField.Powerlock[1].ar_ApparentPower[0]	, 1, 1); 
// eDataMappingVarNames.powermonitor_OutputField_Powerlock_2_ar_ApparentPower_AVG: 				st_Variable:= IotExtractType(monitor.powermonitor.OutputField.Powerlock[2].ar_ApparentPower[0]	, 1, 1); 
// eDataMappingVarNames.powermonitor_OutputField_Powerlock_3_ar_ApparentPower_AVG: 				st_Variable:= IotExtractType(monitor.powermonitor.OutputField.Powerlock[3].ar_ApparentPower[0]	, 1, 1); 
// eDataMappingVarNames.powermonitor_OutputField_Powerlock_1_ar_ApparentPower_L1: 				st_Variable:= IotExtractType(monitor.powermonitor.OutputField.Powerlock[1].ar_ApparentPower[1]		, 1, 1); 
// eDataMappingVarNames.powermonitor_OutputField_Powerlock_2_ar_ApparentPower_L1: 				st_Variable:= IotExtractType(monitor.powermonitor.OutputField.Powerlock[2].ar_ApparentPower[1]		, 1, 1); 
// eDataMappingVarNames.powermonitor_OutputField_Powerlock_3_ar_ApparentPower_L1: 				st_Variable:= IotExtractType(monitor.powermonitor.OutputField.Powerlock[3].ar_ApparentPower[1]		, 1, 1); 
// eDataMappingVarNames.powermonitor_OutputField_Powerlock_1_ar_ApparentPower_L2: 				st_Variable:= IotExtractType(monitor.powermonitor.OutputField.Powerlock[1].ar_ApparentPower[2]		, 1, 1); 
// eDataMappingVarNames.powermonitor_OutputField_Powerlock_2_ar_ApparentPower_L2: 				st_Variable:= IotExtractType(monitor.powermonitor.OutputField.Powerlock[2].ar_ApparentPower[2]		, 1, 1); 
// eDataMappingVarNames.powermonitor_OutputField_Powerlock_3_ar_ApparentPower_L2: 				st_Variable:= IotExtractType(monitor.powermonitor.OutputField.Powerlock[3].ar_ApparentPower[2]		, 1, 1); 
// eDataMappingVarNames.powermonitor_OutputField_Powerlock_1_ar_ApparentPower_L3: 				st_Variable:= IotExtractType(monitor.powermonitor.OutputField.Powerlock[1].ar_ApparentPower[3]		, 1, 1); 
// eDataMappingVarNames.powermonitor_OutputField_Powerlock_2_ar_ApparentPower_L3: 				st_Variable:= IotExtractType(monitor.powermonitor.OutputField.Powerlock[2].ar_ApparentPower[3]		, 1, 1); 
// eDataMappingVarNames.powermonitor_OutputField_Powerlock_3_ar_ApparentPower_L3: 				st_Variable:= IotExtractType(monitor.powermonitor.OutputField.Powerlock[3].ar_ApparentPower[3]		, 1, 1); 
// eDataMappingVarNames.powermonitor_OutputField_Powerlock_1_ar_ReactivePower_AVG: 				st_Variable:= IotExtractType(monitor.powermonitor.OutputField.Powerlock[1].ar_ReactivePower[0]	, 1, 1); 
// eDataMappingVarNames.powermonitor_OutputField_Powerlock_2_ar_ReactivePower_AVG: 				st_Variable:= IotExtractType(monitor.powermonitor.OutputField.Powerlock[2].ar_ReactivePower[0]	, 1, 1); 
// eDataMappingVarNames.powermonitor_OutputField_Powerlock_3_ar_ReactivePower_AVG: 				st_Variable:= IotExtractType(monitor.powermonitor.OutputField.Powerlock[3].ar_ReactivePower[0]	, 1, 1); 
// eDataMappingVarNames.powermonitor_OutputField_Powerlock_1_ar_ReactivePower_L1: 				st_Variable:= IotExtractType(monitor.powermonitor.OutputField.Powerlock[1].ar_ReactivePower[1]		, 1, 1); 
// eDataMappingVarNames.powermonitor_OutputField_Powerlock_2_ar_ReactivePower_L1: 				st_Variable:= IotExtractType(monitor.powermonitor.OutputField.Powerlock[2].ar_ReactivePower[1]		, 1, 1); 
// eDataMappingVarNames.powermonitor_OutputField_Powerlock_3_ar_ReactivePower_L1: 				st_Variable:= IotExtractType(monitor.powermonitor.OutputField.Powerlock[3].ar_ReactivePower[1]		, 1, 1); 
// eDataMappingVarNames.powermonitor_OutputField_Powerlock_1_ar_ReactivePower_L2: 				st_Variable:= IotExtractType(monitor.powermonitor.OutputField.Powerlock[1].ar_ReactivePower[2]		, 1, 1); 
// eDataMappingVarNames.powermonitor_OutputField_Powerlock_2_ar_ReactivePower_L2: 				st_Variable:= IotExtractType(monitor.powermonitor.OutputField.Powerlock[2].ar_ReactivePower[2]		, 1, 1); 
// eDataMappingVarNames.powermonitor_OutputField_Powerlock_3_ar_ReactivePower_L2: 				st_Variable:= IotExtractType(monitor.powermonitor.OutputField.Powerlock[3].ar_ReactivePower[2]		, 1, 1); 
// eDataMappingVarNames.powermonitor_OutputField_Powerlock_1_ar_ReactivePower_L3: 				st_Variable:= IotExtractType(monitor.powermonitor.OutputField.Powerlock[1].ar_ReactivePower[3]		, 1, 1); 
// eDataMappingVarNames.powermonitor_OutputField_Powerlock_2_ar_ReactivePower_L3: 				st_Variable:= IotExtractType(monitor.powermonitor.OutputField.Powerlock[2].ar_ReactivePower[3]		, 1, 1); 
// eDataMappingVarNames.powermonitor_OutputField_Powerlock_3_ar_ReactivePower_L3: 				st_Variable:= IotExtractType(monitor.powermonitor.OutputField.Powerlock[3].ar_ReactivePower[3]		, 1, 1); 
// eDataMappingVarNames.powermonitor_OutputField_Powerlock_1_ar_ActivePower_AVG: 				st_Variable:= IotExtractType(monitor.powermonitor.OutputField.Powerlock[1].ar_ActivePower[0]		, 1, 1); 
// eDataMappingVarNames.powermonitor_OutputField_Powerlock_2_ar_ActivePower_AVG: 				st_Variable:= IotExtractType(monitor.powermonitor.OutputField.Powerlock[2].ar_ActivePower[0]		, 1, 1); 
// eDataMappingVarNames.powermonitor_OutputField_Powerlock_3_ar_ActivePower_AVG: 				st_Variable:= IotExtractType(monitor.powermonitor.OutputField.Powerlock[3].ar_ActivePower[0]		, 1, 1); 
// eDataMappingVarNames.powermonitor_OutputField_Powerlock_1_ar_ActivePower_L1: 				st_Variable:= IotExtractType(monitor.powermonitor.OutputField.Powerlock[1].ar_ActivePower[1]		, 1, 1); 
// eDataMappingVarNames.powermonitor_OutputField_Powerlock_2_ar_ActivePower_L1: 				st_Variable:= IotExtractType(monitor.powermonitor.OutputField.Powerlock[2].ar_ActivePower[1]		, 1, 1); 
// eDataMappingVarNames.powermonitor_OutputField_Powerlock_3_ar_ActivePower_L1: 				st_Variable:= IotExtractType(monitor.powermonitor.OutputField.Powerlock[3].ar_ActivePower[1]		, 1, 1); 
// eDataMappingVarNames.powermonitor_OutputField_Powerlock_1_ar_ActivePower_L2: 				st_Variable:= IotExtractType(monitor.powermonitor.OutputField.Powerlock[1].ar_ActivePower[2]		, 1, 1); 
// eDataMappingVarNames.powermonitor_OutputField_Powerlock_2_ar_ActivePower_L2: 				st_Variable:= IotExtractType(monitor.powermonitor.OutputField.Powerlock[2].ar_ActivePower[2]		, 1, 1); 
// eDataMappingVarNames.powermonitor_OutputField_Powerlock_3_ar_ActivePower_L2: 				st_Variable:= IotExtractType(monitor.powermonitor.OutputField.Powerlock[3].ar_ActivePower[2]		, 1, 1); 
// eDataMappingVarNames.powermonitor_OutputField_Powerlock_1_ar_ActivePower_L3: 				st_Variable:= IotExtractType(monitor.powermonitor.OutputField.Powerlock[1].ar_ActivePower[3]		, 1, 1); 
// eDataMappingVarNames.powermonitor_OutputField_Powerlock_2_ar_ActivePower_L3: 				st_Variable:= IotExtractType(monitor.powermonitor.OutputField.Powerlock[2].ar_ActivePower[3]		, 1, 1); 
// eDataMappingVarNames.powermonitor_OutputField_Powerlock_3_ar_ActivePower_L3: 				st_Variable:= IotExtractType(monitor.powermonitor.OutputField.Powerlock[3].ar_ActivePower[3]		, 1, 1); 
// eDataMappingVarNames.powermonitor_OutputField_Powerlock_1_r_EnergyConsumed: 				st_Variable:= IotExtractType(monitor.powermonitor.OutputField.Powerlock[1].r_EnergyConsumed, 0, 0); 
// eDataMappingVarNames.powermonitor_OutputField_Powerlock_2_r_EnergyConsumed: 				st_Variable:= IotExtractType(monitor.powermonitor.OutputField.Powerlock[2].r_EnergyConsumed, 0, 0); 
// eDataMappingVarNames.powermonitor_OutputField_Powerlock_3_r_EnergyConsumed: 				st_Variable:= IotExtractType(monitor.powermonitor.OutputField.Powerlock[3].r_EnergyConsumed, 0, 0); 
// eDataMappingVarNames.powermonitor_OutputField_Powerlock_1_r_EnergySupplied: 				st_Variable:= IotExtractType(monitor.powermonitor.OutputField.Powerlock[1].r_EnergySupplied, 0, 0); 
// eDataMappingVarNames.powermonitor_OutputField_Powerlock_2_r_EnergySupplied: 				st_Variable:= IotExtractType(monitor.powermonitor.OutputField.Powerlock[2].r_EnergySupplied, 0, 0); 
// eDataMappingVarNames.powermonitor_OutputField_Powerlock_3_r_EnergySupplied: 				st_Variable:= IotExtractType(monitor.powermonitor.OutputField.Powerlock[3].r_EnergySupplied, 0, 0); 
// eDataMappingVarNames.powermonitor_OutputField_Powerlock_1_ar_THD_AVG: 				st_Variable:= IotExtractType(monitor.powermonitor.OutputField.Powerlock[1].ar_THD[0]						, 1, 0); 
// eDataMappingVarNames.powermonitor_OutputField_Powerlock_2_ar_THD_AVG: 				st_Variable:= IotExtractType(monitor.powermonitor.OutputField.Powerlock[2].ar_THD[0]						, 1, 0); 
// eDataMappingVarNames.powermonitor_OutputField_Powerlock_3_ar_THD_AVG: 				st_Variable:= IotExtractType(monitor.powermonitor.OutputField.Powerlock[3].ar_THD[0]						, 1, 0); 
// eDataMappingVarNames.powermonitor_OutputField_Powerlock_1_ar_THD_L1: 				st_Variable:= IotExtractType(monitor.powermonitor.OutputField.Powerlock[1].ar_THD[1]						, 1, 0); 
// eDataMappingVarNames.powermonitor_OutputField_Powerlock_2_ar_THD_L1: 				st_Variable:= IotExtractType(monitor.powermonitor.OutputField.Powerlock[2].ar_THD[1]						, 1, 0); 
// eDataMappingVarNames.powermonitor_OutputField_Powerlock_3_ar_THD_L1: 				st_Variable:= IotExtractType(monitor.powermonitor.OutputField.Powerlock[3].ar_THD[1]						, 1, 0); 
// eDataMappingVarNames.powermonitor_OutputField_Powerlock_1_ar_THD_L2: 				st_Variable:= IotExtractType(monitor.powermonitor.OutputField.Powerlock[1].ar_THD[2]						, 1, 0); 
// eDataMappingVarNames.powermonitor_OutputField_Powerlock_2_ar_THD_L2: 				st_Variable:= IotExtractType(monitor.powermonitor.OutputField.Powerlock[2].ar_THD[2]						, 1, 0); 
// eDataMappingVarNames.powermonitor_OutputField_Powerlock_3_ar_THD_L2: 				st_Variable:= IotExtractType(monitor.powermonitor.OutputField.Powerlock[3].ar_THD[2]						, 1, 0); 
// eDataMappingVarNames.powermonitor_OutputField_Powerlock_1_ar_THD_L3: 				st_Variable:= IotExtractType(monitor.powermonitor.OutputField.Powerlock[1].ar_THD[3]						, 1, 0); 
// eDataMappingVarNames.powermonitor_OutputField_Powerlock_2_ar_THD_L3: 				st_Variable:= IotExtractType(monitor.powermonitor.OutputField.Powerlock[2].ar_THD[3]						, 1, 0); 
// eDataMappingVarNames.powermonitor_OutputField_Powerlock_3_ar_THD_L3: 				st_Variable:= IotExtractType(monitor.powermonitor.OutputField.Powerlock[3].ar_THD[3]						, 1, 0); 
// eDataMappingVarNames.powermonitor_OutputField_Powerlock_1_ar_PowerFactor_AVG: 				st_Variable:= IotExtractType(monitor.powermonitor.OutputField.Powerlock[1].ar_PowerFactor[0]		, 2, 0); 
// eDataMappingVarNames.powermonitor_OutputField_Powerlock_2_ar_PowerFactor_AVG: 				st_Variable:= IotExtractType(monitor.powermonitor.OutputField.Powerlock[2].ar_PowerFactor[0]		, 2, 0); 
// eDataMappingVarNames.powermonitor_OutputField_Powerlock_3_ar_PowerFactor_AVG: 				st_Variable:= IotExtractType(monitor.powermonitor.OutputField.Powerlock[3].ar_PowerFactor[0]		, 2, 0); 
// eDataMappingVarNames.powermonitor_OutputField_Powerlock_1_ar_PowerFactor_L1: 				st_Variable:= IotExtractType(monitor.powermonitor.OutputField.Powerlock[1].ar_PowerFactor[1]		, 2, 0); 
// eDataMappingVarNames.powermonitor_OutputField_Powerlock_2_ar_PowerFactor_L1: 				st_Variable:= IotExtractType(monitor.powermonitor.OutputField.Powerlock[2].ar_PowerFactor[1]		, 2, 0); 
// eDataMappingVarNames.powermonitor_OutputField_Powerlock_3_ar_PowerFactor_L1: 				st_Variable:= IotExtractType(monitor.powermonitor.OutputField.Powerlock[3].ar_PowerFactor[1]		, 2, 0); 
// eDataMappingVarNames.powermonitor_OutputField_Powerlock_1_ar_PowerFactor_L2: 				st_Variable:= IotExtractType(monitor.powermonitor.OutputField.Powerlock[1].ar_PowerFactor[2]		, 2, 0); 
// eDataMappingVarNames.powermonitor_OutputField_Powerlock_2_ar_PowerFactor_L2: 				st_Variable:= IotExtractType(monitor.powermonitor.OutputField.Powerlock[2].ar_PowerFactor[2]		, 2, 0); 
// eDataMappingVarNames.powermonitor_OutputField_Powerlock_3_ar_PowerFactor_L2: 				st_Variable:= IotExtractType(monitor.powermonitor.OutputField.Powerlock[3].ar_PowerFactor[2]		, 2, 0); 
// eDataMappingVarNames.powermonitor_OutputField_Powerlock_1_ar_PowerFactor_L3: 				st_Variable:= IotExtractType(monitor.powermonitor.OutputField.Powerlock[1].ar_PowerFactor[3]		, 2, 0); 
// eDataMappingVarNames.powermonitor_OutputField_Powerlock_2_ar_PowerFactor_L3: 				st_Variable:= IotExtractType(monitor.powermonitor.OutputField.Powerlock[2].ar_PowerFactor[3]		, 2, 0); 
// eDataMappingVarNames.powermonitor_OutputField_Powerlock_3_ar_PowerFactor_L3: 				st_Variable:= IotExtractType(monitor.powermonitor.OutputField.Powerlock[3].ar_PowerFactor[3]		, 2, 0); 
// eDataMappingVarNames.powermonitor_OutputField_Powerlock_1_ar_Current_AVG: 				st_Variable:= IotExtractType(monitor.powermonitor.OutputField.Powerlock[1].ar_Current[0]				, 1, 1); 
// eDataMappingVarNames.powermonitor_OutputField_Powerlock_2_ar_Current_AVG: 				st_Variable:= IotExtractType(monitor.powermonitor.OutputField.Powerlock[2].ar_Current[0]				, 1, 1); 
// eDataMappingVarNames.powermonitor_OutputField_Powerlock_3_ar_Current_AVG: 				st_Variable:= IotExtractType(monitor.powermonitor.OutputField.Powerlock[3].ar_Current[0]				, 1, 1); 
// eDataMappingVarNames.powermonitor_OutputField_Powerlock_1_ar_Current_L1: 				st_Variable:= IotExtractType(monitor.powermonitor.OutputField.Powerlock[1].ar_Current[1]				, 1, 1); 
// eDataMappingVarNames.powermonitor_OutputField_Powerlock_2_ar_Current_L1: 				st_Variable:= IotExtractType(monitor.powermonitor.OutputField.Powerlock[2].ar_Current[1]				, 1, 1); 
// eDataMappingVarNames.powermonitor_OutputField_Powerlock_3_ar_Current_L1: 				st_Variable:= IotExtractType(monitor.powermonitor.OutputField.Powerlock[3].ar_Current[1]				, 1, 1); 
// eDataMappingVarNames.powermonitor_OutputField_Powerlock_1_ar_Current_L2: 				st_Variable:= IotExtractType(monitor.powermonitor.OutputField.Powerlock[1].ar_Current[2]				, 1, 1); 
// eDataMappingVarNames.powermonitor_OutputField_Powerlock_2_ar_Current_L2: 				st_Variable:= IotExtractType(monitor.powermonitor.OutputField.Powerlock[2].ar_Current[2]				, 1, 1); 
// eDataMappingVarNames.powermonitor_OutputField_Powerlock_3_ar_Current_L2: 				st_Variable:= IotExtractType(monitor.powermonitor.OutputField.Powerlock[3].ar_Current[2]				, 1, 1); 
// eDataMappingVarNames.powermonitor_OutputField_Powerlock_1_ar_Current_L3: 				st_Variable:= IotExtractType(monitor.powermonitor.OutputField.Powerlock[1].ar_Current[3]				, 1, 1); 
// eDataMappingVarNames.powermonitor_OutputField_Powerlock_2_ar_Current_L3: 				st_Variable:= IotExtractType(monitor.powermonitor.OutputField.Powerlock[2].ar_Current[3]				, 1, 1); 
// eDataMappingVarNames.powermonitor_OutputField_Powerlock_3_ar_Current_L3: 				st_Variable:= IotExtractType(monitor.powermonitor.OutputField.Powerlock[3].ar_Current[3]				, 1, 1); 
// eDataMappingVarNames.powermonitor_OutputField_Powerlock_1_ar_Current_N: 				st_Variable:= IotExtractType(monitor.powermonitor.OutputField.Powerlock[1].ar_Current[4]				, 1, 1); 
// eDataMappingVarNames.powermonitor_OutputField_Powerlock_2_ar_Current_N: 				st_Variable:= IotExtractType(monitor.powermonitor.OutputField.Powerlock[2].ar_Current[4]				, 1, 1); 
// eDataMappingVarNames.powermonitor_OutputField_Powerlock_3_ar_Current_N: 				st_Variable:= IotExtractType(monitor.powermonitor.OutputField.Powerlock[3].ar_Current[4]				, 1, 1); 
// eDataMappingVarNames.powermonitor_OutputField_Powerlock_1_r_CurrentUnbalance: 				st_Variable:= IotExtractType(monitor.powermonitor.OutputField.Powerlock[1].r_CurrentUnbalance, 0, 0); 
// eDataMappingVarNames.powermonitor_OutputField_Powerlock_2_r_CurrentUnbalance: 				st_Variable:= IotExtractType(monitor.powermonitor.OutputField.Powerlock[2].r_CurrentUnbalance, 0, 0); 
// eDataMappingVarNames.powermonitor_OutputField_Powerlock_3_r_CurrentUnbalance: 				st_Variable:= IotExtractType(monitor.powermonitor.OutputField.Powerlock[3].r_CurrentUnbalance, 0, 0); 
// eDataMappingVarNames.powermonitor_InternalSupply_ar_ApparentPower_AVG: 				st_Variable:= IotExtractType(monitor.powermonitor.InternalSupply.ar_ApparentPower[0], 2, 0); 
// eDataMappingVarNames.powermonitor_InternalSupply_ar_ApparentPower_L1: 				st_Variable:= IotExtractType(monitor.powermonitor.InternalSupply.ar_ApparentPower[1], 2, 0); 
// eDataMappingVarNames.powermonitor_InternalSupply_ar_ApparentPower_L2: 				st_Variable:= IotExtractType(monitor.powermonitor.InternalSupply.ar_ApparentPower[2], 2, 0); 
// eDataMappingVarNames.powermonitor_InternalSupply_ar_ApparentPower_L3: 				st_Variable:= IotExtractType(monitor.powermonitor.InternalSupply.ar_ApparentPower[3], 2, 0); 
// eDataMappingVarNames.powermonitor_InternalSupply_ar_ReactivePower_AVG: 				st_Variable:= IotExtractType(monitor.powermonitor.InternalSupply.ar_ReactivePower[0], 2, 0); 
// eDataMappingVarNames.powermonitor_InternalSupply_ar_ReactivePower_L1: 				st_Variable:= IotExtractType(monitor.powermonitor.InternalSupply.ar_ReactivePower[1], 2, 0); 
// eDataMappingVarNames.powermonitor_InternalSupply_ar_ReactivePower_L2: 				st_Variable:= IotExtractType(monitor.powermonitor.InternalSupply.ar_ReactivePower[2], 2, 0); 
// eDataMappingVarNames.powermonitor_InternalSupply_ar_ReactivePower_L3: 				st_Variable:= IotExtractType(monitor.powermonitor.InternalSupply.ar_ReactivePower[3], 2, 0); 
// eDataMappingVarNames.powermonitor_InternalSupply_ar_ActivePower_AVG: 				st_Variable:= IotExtractType(monitor.powermonitor.InternalSupply.ar_ActivePower[0], 2, 0); 
// eDataMappingVarNames.powermonitor_InternalSupply_ar_ActivePower_L1: 				st_Variable:= IotExtractType(monitor.powermonitor.InternalSupply.ar_ActivePower[1], 2, 0); 
// eDataMappingVarNames.powermonitor_InternalSupply_ar_ActivePower_L2: 				st_Variable:= IotExtractType(monitor.powermonitor.InternalSupply.ar_ActivePower[2], 2, 0); 
// eDataMappingVarNames.powermonitor_InternalSupply_ar_ActivePower_L3: 				st_Variable:= IotExtractType(monitor.powermonitor.InternalSupply.ar_ActivePower[3], 2, 0); 
// eDataMappingVarNames.powermonitor_InternalSupply_r_EnergyConsumed: 				st_Variable:= IotExtractType(monitor.powermonitor.InternalSupply.r_EnergyConsumed, 0, 0); 
// eDataMappingVarNames.powermonitor_InternalSupply_r_EnergySupplied: 				st_Variable:= IotExtractType(monitor.powermonitor.InternalSupply.r_EnergySupplied, 0, 0); 
// eDataMappingVarNames.powermonitor_InternalSupply_ar_THD_AVG: 				st_Variable:= IotExtractType(monitor.powermonitor.InternalSupply.ar_THD[0], 1, 0); 
// eDataMappingVarNames.powermonitor_InternalSupply_ar_THD_L1: 				st_Variable:= IotExtractType(monitor.powermonitor.InternalSupply.ar_THD[1], 1, 0); 
// eDataMappingVarNames.powermonitor_InternalSupply_ar_THD_L2: 				st_Variable:= IotExtractType(monitor.powermonitor.InternalSupply.ar_THD[2], 1, 0); 
// eDataMappingVarNames.powermonitor_InternalSupply_ar_THD_L3: 				st_Variable:= IotExtractType(monitor.powermonitor.InternalSupply.ar_THD[3], 1, 0); 
// eDataMappingVarNames.powermonitor_InternalSupply_ar_PowerFactor_AVG: 				st_Variable:= IotExtractType(monitor.powermonitor.InternalSupply.ar_PowerFactor[0], 2, 0); 
// eDataMappingVarNames.powermonitor_InternalSupply_ar_PowerFactor_L1: 				st_Variable:= IotExtractType(monitor.powermonitor.InternalSupply.ar_PowerFactor[1], 2, 0); 
// eDataMappingVarNames.powermonitor_InternalSupply_ar_PowerFactor_L2: 				st_Variable:= IotExtractType(monitor.powermonitor.InternalSupply.ar_PowerFactor[2], 2, 0); 
// eDataMappingVarNames.powermonitor_InternalSupply_ar_PowerFactor_L3: 				st_Variable:= IotExtractType(monitor.powermonitor.InternalSupply.ar_PowerFactor[3], 2, 0); 
// eDataMappingVarNames.powermonitor_InternalSupply_ar_Current_AVG: 				st_Variable:= IotExtractType(monitor.powermonitor.InternalSupply.ar_Current[0], 1, 1); 
// eDataMappingVarNames.powermonitor_InternalSupply_ar_Current_L1: 				st_Variable:= IotExtractType(monitor.powermonitor.InternalSupply.ar_Current[1], 1, 1); 
// eDataMappingVarNames.powermonitor_InternalSupply_ar_Current_L2: 				st_Variable:= IotExtractType(monitor.powermonitor.InternalSupply.ar_Current[2], 1, 1); 
// eDataMappingVarNames.powermonitor_InternalSupply_ar_Current_L3: 				st_Variable:= IotExtractType(monitor.powermonitor.InternalSupply.ar_Current[3], 1, 1); 
// eDataMappingVarNames.powermonitor_InternalSupply_ar_Current_N: 				st_Variable:= IotExtractType(monitor.powermonitor.InternalSupply.ar_Current[4]	  , 1, 1); 
// eDataMappingVarNames.powermonitor_InternalSupply_r_CurrentUnbalance: 				st_Variable:= IotExtractType(monitor.powermonitor.InternalSupply.r_CurrentUnbalance, 1, 0); 
// eDataMappingVarNames.powermonitor_BESS_e_ACrotationStatus: 				st_Variable:= IotExtractType(monitor.powermonitor.BESS.e_ACrotationStatus, 0, 0); 
// eDataMappingVarNames.powermonitor_BESS_ar_Current_AVG: 				st_Variable:= IotExtractType(monitor.powermonitor.BESS.ar_Current[0], 1, 1); 
// eDataMappingVarNames.powermonitor_BESS_ar_Current_L1: 				st_Variable:= IotExtractType(monitor.powermonitor.BESS.ar_Current[1], 1, 1); 
// eDataMappingVarNames.powermonitor_BESS_ar_Current_L2: 				st_Variable:= IotExtractType(monitor.powermonitor.BESS.ar_Current[2], 1, 1); 
// eDataMappingVarNames.powermonitor_BESS_ar_Current_L3: 				st_Variable:= IotExtractType(monitor.powermonitor.BESS.ar_Current[3], 1, 1); 
// eDataMappingVarNames.powermonitor_BESS_ar_Current_N: 				st_Variable:= IotExtractType(monitor.powermonitor.BESS.ar_Current[4], 1, 1); 
// eDataMappingVarNames.powermonitor_BESS_r_LineVoltage: 				st_Variable:= IotExtractType(monitor.powermonitor.BESS.r_LineVoltage, 1, 1); 
// eDataMappingVarNames.powermonitor_BESS_r_Frequency: 				st_Variable:= IotExtractType(monitor.powermonitor.BESS.r_Frequency, 2, 1); 
// eDataMappingVarNames.powermonitor_BESS_r_currentUnbalance: 				st_Variable:= IotExtractType(monitor.powermonitor.BESS.r_currentUnbalance, 1, 0); 
// eDataMappingVarNames.powermonitor_BESS_r_ApparentPower: 				st_Variable:= IotExtractType(monitor.powermonitor.BESS.r_ApparentPower	, 1, 1); 
// eDataMappingVarNames.powermonitor_BESS_r_ReactivePower: 				st_Variable:= IotExtractType(monitor.powermonitor.BESS.r_ReactivePower	, 1, 1); 
// eDataMappingVarNames.powermonitor_BESS_r_ActivePower: 				st_Variable:= IotExtractType(monitor.powermonitor.BESS.r_ActivePower		, 1, 1); 
// eDataMappingVarNames.powermonitor_BESS_r_EnergyConsumed: 				st_Variable:= IotExtractType(monitor.powermonitor.BESS.r_EnergyConsumed, 0, 0); 
// eDataMappingVarNames.powermonitor_BESS_r_EnergySupplied: 				st_Variable:= IotExtractType(monitor.powermonitor.BESS.r_EnergySupplied, 0, 0); 
// eDataMappingVarNames.powermonitor_BESS_r_PowerFactor: 				st_Variable:= IotExtractType(monitor.powermonitor.BESS.r_PowerFactor, 2, 0); 
// eDataMappingVarNames.powermonitor_events_b_MBCommWarning: 				st_Variable:= IotExtractType(monitor.powermonitor.events.b_MBCommWarning, 0, 0); 
// eDataMappingVarNames.powermonitor_events_b_MBCommError: 				st_Variable:= IotExtractType(monitor.powermonitor.events.b_MBCommError, 0, 0); 
// eDataMappingVarNames.powermonitor_events_b_MBTimeoutWarning: 				st_Variable:= IotExtractType(monitor.powermonitor.events.b_MBTimeoutWarning, 0, 0); 
